(* IEC 61131-3 sources: SmartHomeNew/SmartHomeNew-main/snapshots/clean_build_2026_04_15, 26 files *)

(* ---- E_System_Root_Cause.dut ---- *)
TYPE E_System_Root_Cause :
(
    ROOT_NONE,
    ROOT_FIRE,
    ROOT_GAS_LEAK,
    ROOT_CO_WARNING,
    ROOT_CO_CRITICAL,
    ROOT_WATER_LEAK,
    ROOT_IO_OFFLINE,
    ROOT_COMM_FAULT,
    ROOT_SENSOR_FAULT,
    ROOT_SUBSYSTEM_FAULT,
    ROOT_WATCHDOG_FAULT
);
END_TYPE

(* ---- E_VENTILATION_LOCATION.dut ---- *)
{attribute 'strict'}
TYPE E_VENTILATION_LOCATION :
(
  VENT_LOCATION_NONE := 0,
  VENT_LOCATION_BASEMENT_GAME_ROOM := 1,
  VENT_LOCATION_BASEMENT_GYM := 2,
  VENT_LOCATION_BASEMENT_BOILER_ROOM := 3,
  VENT_LOCATION_BATHROOM_1F := 4,
  VENT_LOCATION_BATHROOM_2F := 5,
  VENT_LOCATION_MASTER_BATHROOM := 6,
  VENT_LOCATION_LAUNDRY := 7,
  VENT_LOCATION_KITCHEN := 8
) USINT;
END_TYPE

(* ---- ST_Heating_Command_V2.dut ---- *)
TYPE ST_Heating_Command_V2 : STRUCT
    Valve_Position_Setpoint : REAL;
END_STRUCT
END_TYPE

(* ---- ST_Lighting_Command_V2.dut ---- *)
TYPE ST_Lighting_Command_V2 : STRUCT
    Brightness_Setpoint : REAL;
END_STRUCT
END_TYPE

(* ---- ST_Maintenance_Access_Config.dut ---- *)
{attribute 'pack_mode' := '1'}
TYPE ST_Maintenance_Access_Config :
STRUCT
    maintenance_enabled : BOOL := FALSE;
    max_duration_minutes : UDINT := 60;
    requires_two_person : BOOL := TRUE;
    access_level_required : BYTE := 2;
END_STRUCT
END_TYPE

(* ---- ST_System_Diagnostics.dut ---- *)
{attribute 'pack_mode' := '1'}
TYPE ST_System_Diagnostics :
STRUCT
    Freeze_Hardware_Event_Pending : BOOL;
    Freeze_Hardware_Event_Text : STRING(200);
    Backup_Pump_Fault : BOOL;
    Electric_Heater_Fault : BOOL;
    Backup_Pump_Recovered_After_Retry : BOOL;
    Electric_Heater_Recovered_After_Retry : BOOL;
    Backup_Pump_Out_Of_Service : BOOL;
    Electric_Heater_Out_Of_Service : BOOL;

    Pump_Exercise_Active : BOOL;
    Pump_Exercise_Failed : BOOL;
    Pump_Exercise_Last_Equipment : STRING(80);
    Pump_Exercise_Last_Result : STRING(120);
    Pump_Exercise_No_Feedback_Count : INT;
    Manifold_Pump_Exercise_Count : ARRAY[1..GVL_CONSTANTS.C_MAX_MANIFOLDS] OF UDINT;
    DHW_Heating_Pump_Exercise_Count : UDINT;
    DHW_Circ_Pump_Exercise_Count : UDINT;
    Backup_Pump_Exercise_Count : UDINT;
    Pump_Exercise_Event_Seq : UDINT;
    Pump_Exercise_Journal_1 : STRING(200);
    Pump_Exercise_Journal_2 : STRING(200);
    Pump_Exercise_Journal_3 : STRING(200);
    Pump_Exercise_Journal_Last_Seq : UDINT;

    Pump_Maintenance_Required : BOOL;
    Pump_Maintenance_Warning : BOOL;

    Manifold_Pump_Out_Of_Service : ARRAY[1..GVL_CONSTANTS.C_MAX_MANIFOLDS] OF BOOL;
    DHW_Heating_Pump_Out_Of_Service : BOOL;
    DHW_Circ_Pump_Out_Of_Service : BOOL;

    Maintenance_Last_Action : STRING(120);
    Operator_Action_Blocked : BOOL;
    Operator_Block_Reason : STRING(160);
    Operator_Last_Forbidden_Action : STRING(160);
    Operator_Journal_1 : STRING(200);
    Operator_Journal_2 : STRING(200);
    Operator_Journal_3 : STRING(200);
    Operator_Journal_Event_Seq : UDINT;
    Operator_Journal_Last_Seq : UDINT;

    Dangerous_Action_Pending_Confirm : BOOL;
    Dangerous_Action_Confirm_Text : STRING(160);
    Dangerous_Action_Confirm_Deadline_MS : UDINT;
    User_Access_Level_Active : INT;
    User_Access_Denied : BOOL;
    User_Access_Deny_Reason : STRING(160);

    Valve_Test_Mode_Active : BOOL;
    Valve_Test_Deadline_MS : UDINT;
    Valve_Test_Remaining_MS : UDINT;
    Valve_Test_Validation_OK : BOOL;
    Valve_Test_Validation_Text : STRING(160);
    Valve_Test_Forced_Close : BOOL;

    Water_Valve_Test_Mode_Active : BOOL;
    Water_Valve_Test_Deadline_MS : UDINT;
    Water_Valve_Test_Remaining_MS : UDINT;
    Water_Valve_Test_Validation_OK : BOOL;
    Water_Valve_Test_Validation_Text : STRING(160);
    Water_Valve_Test_Forced_Close : BOOL;
    Gas_Valve_Test_Mode_Active : BOOL;
    Gas_Valve_Test_Deadline_MS : UDINT;
    Gas_Valve_Test_Remaining_MS : UDINT;
    Gas_Valve_Test_Validation_OK : BOOL;
    Gas_Valve_Test_Validation_Text : STRING(160);
    Gas_Valve_Test_Forced_Close : BOOL;

    Active_Leak_Sensor_Index : INT;
    Active_Gas_Sensor_Index : INT;
    Active_Leak_Zone_Name : STRING(80);
    Active_Gas_Zone_Name : STRING(80);
    Water_Valve_Test_Context : STRING(160);
    Gas_Valve_Test_Context : STRING(160);

    Water_Recovery_Target_Zone_Index : INT;
    Gas_Recovery_Target_Zone_Index : INT;
    Water_Recovery_Selective_Allowed : BOOL;
    Gas_Recovery_Selective_Allowed : BOOL;
    Water_Recovery_Selective_Text : STRING(160);
    Gas_Recovery_Selective_Text : STRING(160);
    Water_Recovery_Physical_Active : BOOL;
    Water_Recovery_Physical_Zone_Name : STRING(80);

    Water_Zone_Open_Fault : ARRAY[1..32] OF BOOL;
    Water_Zone_Close_Fault : ARRAY[1..32] OF BOOL;
    Water_Valve_Exercise_Last_Zone : INT;
    Water_Valve_Exercise_Last_Result : STRING(160);
    Water_Zone_Critical_Close_Fault : ARRAY[1..32] OF BOOL;
    Water_Close_Fault_Active : BOOL;
    Water_Close_Fault_Zone_Name : STRING(80);
    Water_Close_Fault_Text : STRING(200);
    Water_Zone_Close_Retry_Active : ARRAY[1..32] OF BOOL;
    Water_Zone_Close_Retry_Count : ARRAY[1..32] OF INT;
    Water_Zone_Close_Recovered_After_Retry : ARRAY[1..32] OF BOOL;
    Water_Localization_Failed : BOOL;
    Water_Main_Shutdown_Recommended : BOOL;
    Water_Escalation_Text : STRING(200);
    Alarm_Event_Pulse : BOOL;
    Alarm_Event_Code : UDINT;
    Alarm_Event_Value : REAL;
    Sensor_Fault : BOOL;
    IO_Offline : BOOL;
    Subsystem_Degraded : BOOL;

END_STRUCT
END_TYPE

(* ---- ST_Ventilation_Command_V2.dut ---- *)
TYPE ST_Ventilation_Command_V2 : STRUCT
    Fan_Speed_Setpoint : REAL;
END_STRUCT
END_TYPE

(* ---- GVL_CONFIG.gvl ---- *)
{attribute 'qualified_only'}
VAR_GLOBAL
    // Subsystem Configurations
    G_Heating_Config : ST_Heating_Config; // Настройки системы отопления
    G_Ventilation_Config : ST_Ventilation_Config; // Настройки системы вентиляции
    G_DHW_Config : ST_DHW_Config; // Настройки горячего водоснабжения
    G_Security_Config : ST_Security_Global_Config; // Настройки системы безопасности
    G_Flood_Config : ST_Flood_Config; // Настройки системы защиты от протечек

    // HMI Configurations
    G_HMI_FloorHeating_Configs : ARRAY[1..8] OF ST_FloorHeating_Circuit_Config; // Конфигурации контуров теплого пола
    G_Wet_Zone_Map : ARRAY[1..32] OF BOOL; // Карта мокрых зон (TRUE = мокрая зона)
    G_HMI_Tariff_Settings : ST_Tariff_Config; // Настройки тарифов
    G_HMI_Vent_Global_Config : ST_Ventilation_Global_Config; // Глобальные настройки вентиляции
    G_HMI_Vent_Unit_Configs : ARRAY[1..GVL_CONSTANTS.C_MAX_VENT_UNITS] OF ST_Ventilation_Unit_Config; // Конфигурации отдельных вентустановок
    G_HMI_Scenario_Configs : ARRAY[1..GVL_CONSTANTS.C_MAX_SCENARIOS] OF ST_Scenario_Config; // Конфигурации сценариев
    G_HMI_Outdoor_Configs : ARRAY[1..GVL_CONSTANTS.C_MAX_OUTDOOR_ZONES] OF ST_Outdoor_Zone_Config; // Конфигурации зон уличного освещения
    G_HMI_Flood_Config : ST_Flood_Global_Config; // Глобальные настройки защиты от протечек
    G_HMI_Gas_Config : ST_Gas_Valve_Configuration; // Конфигурация системы газового контроля
    G_HMI_Sensor_Calibrations : ARRAY[1..GVL_CONSTANTS.C_MAX_CALIBRATIONS] OF ST_Sensor_Calibration_Record; // Данные калибровки датчиков
    G_HMI_User_Rules : ARRAY[1..GVL_CONSTANTS.C_MAX_RULES] OF ST_User_Rule; // Пользовательские правила (Rule Engine)

    // Конфигурация тестирования клапанов
    G_Valve_Test_Config : ARRAY[1..GVL_CONSTANTS.C_MAX_MANIFOLDS] OF ST_Valve_Test_Config;

    // HMI Commands & States
    G_HMI_Cleaning_Mode_Active : ARRAY[1..GVL_CONSTANTS.C_MAX_CLEANING_MODES] OF BOOL; // Режим уборки активен
    G_HMI_Cleaning_Mode_TimeLeft : ARRAY[1..GVL_CONSTANTS.C_MAX_CLEANING_MODES] OF UINT; // Оставшееся время режима уборки
    G_HMI_Admin_2FA_Enabled : BOOL := FALSE; // Включена ли 2FA для ADMIN
    G_HMI_Current_Operator_Factor2_Done : BOOL; // Второй фактор пройден
    G_HMI_Current_Operator_ID : STRING(10); // ID текущего оператора
    G_HMI_Manual_Gas_Valve_Open : BOOL; // Ручное открытие газового клапана
    G_HMI_Manual_Gas_Valve_Time : UDINT := 5; // Время ручного открытия
    G_HMI_Manual_Gas_Valve_TimeLeft : UDINT; // Оставшееся время ручного открытия
    G_HMI_Apply_Settings : BOOL; // Команда: Применить настройки
    G_HMI_Mute_Alarm : BOOL; // Команда: Временное отключение сирены
    G_HMI_Ack_Alarms : BOOL; // Команда: Квитировать все тревоги

    // Access Control Commands
    G_HMI_Gate_Open_Req : BOOL; // Запрос на открытие въездных ворот
    G_HMI_Wicket_Open_Req : BOOL; // Запрос на открытие калитки
    G_HMI_Lock_1_Open_Req : BOOL; // Разблокировка основного замка
    G_HMI_Lock_1_Close_Req : BOOL; // Блокировка основного замка
    G_HMI_Lock_2_Open_Req : BOOL; // Разблокировка доп. замка
    G_HMI_Lock_2_Close_Req : BOOL; // Блокировка доп. замка

    // HMI Settings
    G_HMI_Language : BYTE := 0; // 0=RU, 1=EN
    G_HMI_Brightness : BYTE := 80;
    G_HMI_Screen_Saver_Timeout : UDINT := 300; // сек

    // Сетевая безопасность
    G_Allowed_IPs : ARRAY[1..GVL_CONSTANTS.C_MAX_ALLOWED_IPS] OF STRING(15) := ['192.168.1.100','192.168.1.101','127.0.0.1','','']; // Разрешенные IP-адреса для шлюза

    G_Backup_Circulation_Pump_In_Service : BOOL := TRUE; // Резервный насос доступен для логики
    G_Electric_Heater_In_Service : BOOL := TRUE; // Электронагреватель доступен для логики
    G_Freeze_Hardware_Retry_Count : INT := 2; // Количество повторных попыток для anti-freeze hardware
    G_Freeze_Hardware_Retry_Delay_MS : UDINT := 5000; // Задержка между попытками повторного пуска
    G_Pump_Exercise_Enabled : BOOL := TRUE; // Разрешение периодической прокрутки насосов после простоя
    G_Pump_Exercise_Interval_MS : UDINT := 604800000; // 7 суток
    G_Pump_Exercise_Duration_MS : UDINT := 30000; // 30 сек
    G_Manifold_Pump_In_Service : ARRAY[1..GVL_CONSTANTS.C_MAX_MANIFOLDS] OF BOOL := [TRUE, TRUE, TRUE, TRUE, TRUE];
    G_DHW_Heating_Pump_In_Service : BOOL := TRUE;
    G_DHW_Circ_Pump_In_Service : BOOL := TRUE;
    G_Water_Valve_Exercise_Enabled : BOOL := TRUE;
    G_Water_Valve_Exercise_Interval_MS : UDINT := 604800000;
    G_Water_Valve_Exercise_Duration_MS : UDINT := 15000;
    G_Water_Valve_Exercise_Window_Start : TOD := TOD#04:00;
    G_Water_Valve_Exercise_Window_End : TOD := TOD#05:00;
    G_Water_Valve_Close_Retry_Count : INT := 2;
    G_Water_Valve_Close_Retry_Delay_MS : UDINT := 3000;
    // IO Mapping
    G_FloorTemp_Map : ARRAY[1..8] OF INT := [1, 2, 3, 4, 5, 6, 7, 8];
    G_RoomTemp_Map : ARRAY[1..16] OF INT := [1, 2, 3, 4, 5, 6, 7, 8, 9, 10, 11, 12, 13, 14, 15, 16];
    G_Door_Map : ARRAY[1..GVL_CONSTANTS.C_MAX_DOOR_SENSORS] OF INT := [1, 2, 3, 4, 5, 6, 7, 8];
    G_Window_Map : ARRAY[1..16] OF INT := [9, 10, 11, 12, 13, 14, 15, 16, 17, 18, 19, 20, 21, 22, 23, 24];

    // Evacuation config
    C_MAX_LIGHT_ZONES : INT := 32; // fallback if not defined elsewhere
    G_Evac_Exit_Zones : ARRAY[1..32] OF BOOL; // зоны-выходы (TRUE = выход)
    G_Evac_Smoke_Zone_Map : ARRAY[1..GVL_CONSTANTS.C_MAX_SMOKE_SENSORS] OF INT; // Привязка дымовых датчиков к зонам эвакуации
    G_Evac_Leak_Zone_Map : ARRAY[1..GVL_CONSTANTS.C_MAX_FLOOD_SENSORS] OF INT; // Привязка датчиков протечки к зонам эвакуации
    G_Evac_Gas_Zone_Map : ARRAY[1..GVL_CONSTANTS.C_MAX_METHANE_SENSORS] OF INT; // Привязка газовых датчиков к зонам эвакуации
    G_Evac_Zone_Names : ARRAY[1..32] OF STRING(80); // Человекочитаемые имена зон (помещения/крыло/этаж/сторона)

END_VAR

VAR_GLOBAL CONSTANT
    C_MS_PER_SEC    : UDINT := GVL_CONSTANTS.C_MS_IN_SECOND; // Миллисекунд в секунде
    C_SEC_PER_MIN   : UDINT := 60; // Секунд в минуте
    C_MIN_PER_HOUR  : UDINT := 60; // Минут в часе
    C_MS_PER_MIN    : UDINT := GVL_CONSTANTS.C_MS_IN_MINUTE; // Миллисекунд в минуте
    C_MAX_RULES     : INT := 20; // Максимальное количество пользовательских правил
    C_ZONE_COUNT    : BYTE := 18; // Общее количество зон в системе

    // Коды ошибок
    ERR_PRESSURE_OUT_OF_RANGE : UDINT := 16#E004;
    ERR_HIGH_DELTA_T : UDINT := 16#E005;
    ERR_BOILER_OFFLINE : UDINT := 16#E006;
    ERR_BOILER_GENERAL_FAULT : UDINT := 16#E007;
    ERR_BOILER_NO_FLAME : UDINT := 16#E008;
    ERR_PUMP_NO_CURRENT : UDINT := 16#E009;
    ERR_PUMP_UNDERCURRENT : UDINT := 16#E00A;
    ERR_PUMP_OVERCURRENT : UDINT := 16#E00B;
    ERR_DELTA_T_LOW : UDINT := 16#E00C;
    ERR_DELTA_T_HIGH : UDINT := 16#E00D;
    ERR_DHW_IO_OFFLINE : UDINT := 16#E00E;
    ERR_DHW_TEMP_SENSOR_FAULT : UDINT := 16#E00F;
    ERR_DHW_PRESSURE_OUT_OF_RANGE : UDINT := 16#E010;
    ERR_DHW_PRESSURE_SENSOR_FAULT : UDINT := 16#E011;
END_VAR

(* ---- GVL_HEALTH_BRIDGE.gvl ---- *)
{attribute 'qualified_only'}
VAR_GLOBAL
    G_Smoke_Detected : BOOL;
    G_Gas_Detected : BOOL;
    G_Leak_Detected : BOOL;
    G_Leak_Warning_Level : BOOL;
    G_CO_Warning_Level : BOOL;
    G_CO_Alarm_Level : BOOL;
    G_Last_Fault_Event_Text : STRING(255);
END_VAR

(* ---- GVL_HEALTH_BRIDGE.st ---- *)
VAR_GLOBAL
    G_Smoke_Detected      : BOOL := FALSE;
    G_Gas_Detected        : BOOL := FALSE;
    G_CO_Warning_Level    : BOOL := FALSE;
    G_CO_Alarm_Level      : BOOL := FALSE;
    G_Leak_Detected       : BOOL := FALSE;
    G_Leak_Warning_Level  : BOOL := FALSE;

    G_Last_Fault_Event_Text : STRING(200) := '';
END_VAR

(* ---- FB_Astro_Timer.st ---- *)
FUNCTION_BLOCK FB_Astro_Timer
VAR_INPUT
    VI_System_Time_MS : UDINT;
    VI_Latitude : REAL := 55.75; // Москва (по умолчанию)
    VI_Longitude : REAL := 37.61;
    VI_Timezone : REAL := 3.0; // UTC+3
    VI_Day_Of_Year : UINT; // День года (1-365)
END_VAR
// >>> SYNC_TEST_MARKER_002 <<<
VAR_OUTPUT
    VO_Sunset_Time : TOD;
    VO_Sunrise_Time : TOD;
    VO_Is_Night : BOOL;
    VO_Current_TOD : TOD; // Текущее время суток
END_VAR
VAR
    L_Current_TOD : TOD;
    L_Pi : REAL := 3.14159265359;
    L_Rad : REAL := 3.14159265359 / 180.0;
    L_Deg : REAL := 180.0 / 3.14159265359;
    L_B : REAL;
    L_EoT : REAL;
    L_Declination : REAL;
    L_Cos_Omega : REAL;
    L_Omega : REAL;
    L_Sunrise_Local : REAL;
    L_Sunset_Local : REAL;
END_VAR

L_Current_TOD := GVL_STATUS.G_Current_TOD;
VO_Current_TOD := L_Current_TOD;

// Equation of Time (EoT) in minutes
L_B := 360.0 / 365.0 * TO_REAL(VI_Day_Of_Year - 81) * L_Rad;
L_EoT := 9.87 * SIN(2.0 * L_B) - 7.53 * COS(L_B) - 1.5 * SIN(L_B);

// Solar Declination in degrees
L_Declination := 23.45 * SIN(360.0 / 365.0 * TO_REAL(VI_Day_Of_Year + 284) * L_Rad);

// Hour angle
L_Cos_Omega := -TAN(VI_Latitude * L_Rad) * TAN(L_Declination * L_Rad);

IF L_Cos_Omega > 1.0 THEN
    L_Cos_Omega := 1.0; // Polar night
ELSIF L_Cos_Omega < -1.0 THEN
    L_Cos_Omega := -1.0; // Polar day
END_IF;

L_Omega := ACOS(L_Cos_Omega) * L_Deg;

// Sunrise and Sunset in local time (hours)
L_Sunrise_Local := 12.0 - (L_Omega / 15.0) - (L_EoT / 60.0) + (VI_Timezone * 15.0 - VI_Longitude) / 15.0;
L_Sunset_Local := 12.0 + (L_Omega / 15.0) - (L_EoT / 60.0) + (VI_Timezone * 15.0 - VI_Longitude) / 15.0;

// Handle bounds
IF L_Sunrise_Local < 0.0 THEN L_Sunrise_Local := L_Sunrise_Local + 24.0; END_IF;
IF L_Sunrise_Local >= 24.0 THEN L_Sunrise_Local := L_Sunrise_Local - 24.0; END_IF;
IF L_Sunset_Local < 0.0 THEN L_Sunset_Local := L_Sunset_Local + 24.0; END_IF;
IF L_Sunset_Local >= 24.0 THEN L_Sunset_Local := L_Sunset_Local - 24.0; END_IF;

// Конвертация в TOD
VO_Sunrise_Time := TO_TOD(TO_UDINT(L_Sunrise_Local * 3600000.0));
VO_Sunset_Time := TO_TOD(TO_UDINT(L_Sunset_Local * 3600000.0));

// ТЗ 15.2: Закат + 30 мин / Рассвет - 30 мин
VO_Is_Night := (L_Current_TOD > (VO_Sunset_Time + T#30m)) OR (L_Current_TOD < (VO_Sunrise_Time - T#30m));
// >>> SYNC_TEST_MARKER_FORCE <<<
// >>> BULK_SYNC_ANCHOR: FB_Astro_Timer <<<

(* ---- FB_DHW_Manager.st ---- *)
FUNCTION_BLOCK FB_DHW_Manager
VAR_INPUT
    VI_System_Time_MS : UDINT; // Системное время (мс)
    VI_Current_TOD : TOD; // Текущее время суток
    VI_IsActivePLC : BOOL; // Флаг: Данный ПЛК является ведущим
    VI_Temp : REAL; // Текущая температура воды в бойлере (°C)
    VI_Pressure : REAL; // Текущее давление в системе ГВС (бар)
    VI_Config : ST_DHW_Config; // Конфигурация системы ГВС (уставки, расписание)
    VI_Current_Day_Of_Week : UINT; // Текущий день недели (1-7)
    VI_Reset_Errors : BOOL; // Сброс ошибок
    VI_Emergency_Stop : BOOL; // Агрегированный аварийный стоп от подсистемы безопасности
    VI_System_Mode : E_System_Operating_Mode; // Агрегированный режим системы
    VI_IO_Modules_Online : ARRAY[1..GVL_CONSTANTS.C_MAX_MODULES] OF BOOL; // Статусы модулей ввода-вывода (только чтение)
END_VAR
// >>> SYNC_TEST_MARKER_001 <<<
VAR_OUTPUT
    VO_Status : ST_DHW_Status; // Сводный статус системы ГВС для HMI
    VO_Heating_Pump : BOOL; // Выход: Управление насосом нагрева (загрузка бойлера)
    VO_Circ_Pump : BOOL; // Выход: Управление насосом рециркуляции ГВС
END_VAR
VAR
    // DHW V2 staging layer
    fbDHWV2Staging : FB_DHW_V2_Staging;
    L_DHW_V2_Command_V2 : ST_DHW_Command_V2;
    L_DHW_V2_State_V2 : ST_DHW_State_V2;
    L_DHW_V2_Shadow_Diff_Found : BOOL;
    L_DHW_V2_Switch_Enabled : BOOL;
    L_DHW_V2_Path_Ready : BOOL;
    L_DHW_Using_Legacy_Fallback : BOOL;
    L_i : INT;
    L_Current_TOD : TOD; // Текущее время суток
    L_Legionella_Active : BOOL; // Флаг активного режима термической дезинфекции (Легионелла)
    L_Legionella_Timer : FB_System_Timer; // Таймер удержания температуры для дезинфекции
    L_Last_Good_Temp : REAL := 55.0; // Последнее достоверное значение температуры (для Fallback)
    L_Legionella_Done_Today : BOOL; // Признак выполнения термодезинфекции в текущие сутки
    L_Last_Legionella_Day : UINT; // День недели последнего сброса/контроля цикла легионеллы
    fbTempValidator : FB_Analog_Validator;
    fbPressValidator : FB_Analog_Validator;
    L_Error_Latched : BOOL;
    L_Error_ID_Latched : WORD;
    L_Policy_Degraded : BOOL;
    L_Policy_Freeze_Protection : BOOL;
    L_Policy_Safe_Stop : BOOL;
    L_Target_Temp_Adjusted : REAL;
END_VAR

IF NOT VI_IsActivePLC THEN RETURN; END_IF;

L_DHW_V2_Shadow_Diff_Found := FALSE;
L_DHW_V2_Switch_Enabled := TRUE;
L_DHW_V2_Path_Ready := FALSE;
L_DHW_Using_Legacy_Fallback := TRUE;

GVL_STATE.G_DHW_IO_Fault := FALSE;
GVL_STATE.G_DHW_Sensor_Fault := FALSE;
GVL_STATE.G_DHW_Subsystem_Degraded := FALSE;

IF VI_Emergency_Stop THEN
    VO_Heating_Pump := FALSE;
    VO_Circ_Pump := FALSE;
    VO_Status.Warning := FALSE;
    VO_Status.Error := TRUE;
    VO_Status.Error_ID := TO_WORD(GVL_CONFIG.ERR_DHW_IO_OFFLINE); // временно используем общий аварийный код до детализации safety-кодов
    VO_Status.Heating_Pump_On := FALSE;
    VO_Status.Circ_Pump_On := FALSE;
    RETURN;
END_IF;

// Фиксация текущего времени
L_Current_TOD := VI_Current_TOD;

// ========================================
// DHW POLICY LAYER
// ========================================
L_Policy_Safe_Stop := (VI_System_Mode = E_System_Operating_Mode.MODE_SAFE_STOP);
L_Policy_Freeze_Protection := (VI_System_Mode = E_System_Operating_Mode.MODE_FREEZE_PROTECTION);
L_Policy_Degraded := (VI_System_Mode = E_System_Operating_Mode.MODE_DEGRADED);
L_Target_Temp_Adjusted := VI_Config.Target_Temp;
IF L_Policy_Degraded THEN
    L_Target_Temp_Adjusted := VI_Config.Target_Temp - VI_Config.Degraded_Target_Delta;
END_IF;

// ========================================
// DHW POLICY OVERRIDE
// ========================================
IF L_Policy_Safe_Stop THEN
    VO_Heating_Pump := FALSE;
    VO_Circ_Pump := FALSE;
    RETURN;
END_IF;

IF L_Policy_Freeze_Protection THEN
    VO_Heating_Pump := FALSE;
    VO_Circ_Pump := FALSE;
    RETURN;
END_IF;

// Сброс признака выполнения термодезинфекции при смене дня.
IF L_Last_Legionella_Day <> VI_Current_Day_Of_Week THEN
    L_Legionella_Done_Today := FALSE;
    L_Last_Legionella_Day := VI_Current_Day_Of_Week;
END_IF;

// Базовый сброс незащёлкнутых статусных флагов на текущий цикл.
// Критические ошибки ниже могут зафиксироваться и завершить выполнение через RETURN.
VO_Status.Warning := FALSE;
VO_Status.Error := FALSE;
VO_Status.Error_ID := 0;

// Сброс ошибок
IF VI_Reset_Errors THEN
    L_Error_Latched := FALSE;
    L_Error_ID_Latched := 0;
END_IF;

// Проверка связи с модулями ввода-вывода
FOR L_i := 1 TO GVL_CONSTANTS.C_MAX_MODULES DO
    IF NOT VI_IO_Modules_Online[L_i] THEN
        L_Error_Latched := TRUE;
        GVL_STATE.G_DHW_IO_Fault := TRUE;
        L_Error_ID_Latched := TO_WORD(GVL_CONFIG.ERR_DHW_IO_OFFLINE); // Потеря связи с модулями ввода-вывода
    END_IF;
END_FOR;

// 1. Обработка неисправностей датчиков и сервисных режимов (ТЗ 7.0)
fbTempValidator(
    VI_Value := VI_Temp,
    VI_Min_Valid := 0.0,
    VI_Max_Valid := 100.0,
    VI_Fallback_Mode := 0,
    VI_Default_Value := 55.0
);

fbPressValidator(
    VI_Value := VI_Pressure,
    VI_Min_Valid := 0.0,
    VI_Max_Valid := 10.0,
    VI_Fallback_Mode := 0
);

VO_Status.Temp := fbTempValidator.VO_Value;
VO_Status.Pressure := fbPressValidator.VO_Value;

// Сохраняем последнее достоверное значение температуры ГВС.
// Используется только для диагностики/сервиса, не для fallback-управления.
IF NOT fbTempValidator.VO_Error THEN
    L_Last_Good_Temp := VO_Status.Temp;
END_IF;

IF fbTempValidator.VO_Error THEN
    GVL_STATE.G_DHW_Sensor_Fault := TRUE;
    L_Error_Latched := TRUE;
    L_Error_ID_Latched := TO_WORD(GVL_CONFIG.ERR_DHW_TEMP_SENSOR_FAULT); // Критическая ошибка датчика температуры
ELSIF (VO_Status.Pressure < 1.0 OR VO_Status.Pressure > 4.0) AND NOT fbPressValidator.VO_Error THEN
    L_Error_Latched := TRUE;
    L_Error_ID_Latched := TO_WORD(GVL_CONFIG.ERR_DHW_PRESSURE_OUT_OF_RANGE); // Давление вне нормы
END_IF;

IF L_Error_Latched THEN
    // Критическая ошибка: переход в безопасное состояние с полной остановкой насосов.
    VO_Heating_Pump := FALSE;
    VO_Circ_Pump := FALSE;
    VO_Status.Warning := FALSE;
    VO_Status.Error := TRUE;
    VO_Status.Error_ID := L_Error_ID_Latched;
    VO_Status.Heating_Pump_On := FALSE;
    VO_Status.Circ_Pump_On := FALSE;
    RETURN;
END_IF;

// Ошибка датчика давления не останавливает ГВС,
// но переводит подсистему в режим предупреждения (degraded mode).
IF fbPressValidator.VO_Error THEN
    GVL_STATE.G_DHW_Sensor_Fault := TRUE;
    GVL_STATE.G_DHW_Subsystem_Degraded := TRUE;
    VO_Status.Warning := TRUE;
    VO_Status.Error := FALSE;
    VO_Status.Error_ID := TO_WORD(GVL_CONFIG.ERR_DHW_PRESSURE_SENSOR_FAULT);
END_IF;

// 2. Логика поддержания температуры воды в бойлере (Нагрев)
// На этом этапе FB уже выполняется только на активном ПЛК.

// Термическая дезинфекция (Легионелла)
IF VI_Config.Anti_Legionella_Enabled
   AND (VI_Current_Day_Of_Week = VI_Config.Anti_Legionella_Day)
   AND (L_Current_TOD >= TOD#02:00)
   AND (L_Current_TOD <= TOD#04:00)
   AND NOT L_Legionella_Done_Today THEN
    L_Legionella_Active := TRUE;
ELSE
    L_Legionella_Active := FALSE;
END_IF;

L_Legionella_Timer(IN := L_Legionella_Active AND VO_Status.Temp >= 70.0, PT := T#30m, VI_System_Time_MS := VI_System_Time_MS);
IF L_Legionella_Timer.Q THEN
    L_Legionella_Active := FALSE; // Дезинфекция завершена
    L_Legionella_Done_Today := TRUE; // Повторно в те же сутки не запускать
END_IF;

// Двухпозиционное регулирование с гистерезисом
IF L_Legionella_Active THEN
    IF VO_Status.Temp < 70.0 THEN
        VO_Heating_Pump := TRUE;
    ELSIF VO_Status.Temp > 72.0 THEN
        VO_Heating_Pump := FALSE;
    END_IF;
ELSE
    IF VO_Status.Temp < (L_Target_Temp_Adjusted - VI_Config.Hysteresis) THEN
        VO_Heating_Pump := TRUE;
    ELSIF VO_Status.Temp > (L_Target_Temp_Adjusted + VI_Config.Hysteresis) THEN
        VO_Heating_Pump := FALSE;
    END_IF;
END_IF;

// 3. Управление циркуляционным насосом ГВС по расписанию
// Рециркуляция обеспечивает мгновенное наличие горячей воды у потребителя
VO_Circ_Pump := SEL(VI_Config.Circulation_Schedule_Enabled AND NOT (VI_Config.Night_Mode_Enabled AND (L_Current_TOD < VI_Config.Circulation_Start OR L_Current_TOD > VI_Config.Circulation_End)), FALSE, TRUE);

// Формирование статусных данных для визуализации.
// К этому моменту статус уже консистентен:
// - Error = критическая ошибка с остановкой ГВС
// - Warning = деградация без остановки
VO_Status.Heating_Pump_On := VO_Heating_Pump;
VO_Status.Circ_Pump_On := VO_Circ_Pump;

// ========================================
// DHW V2 staging execution
// ========================================
fbDHWV2Staging(
    VI_Tank_ID := 1,
    VI_Enable := TRUE,
    VI_Target_Temp := VI_Config.Target_Temp,
    VI_Pump_Enable := VO_Heating_Pump,
    VI_Heating_Priority := FALSE,

    VI_Is_Active := TRUE,
    VI_Tank_Temp := VO_Status.Temp,
    VI_Supply_Temp := VO_Status.Temp,
    VI_Return_Temp := VO_Status.Temp,
    VI_Pump_Actual := VO_Heating_Pump,
    VI_Alarm_Active := VO_Status.Error,

    VO_Command_Shadow => L_DHW_V2_Command_V2,
    VO_State_Shadow => L_DHW_V2_State_V2
);

// ========================================
// DHW V2 staging validation
// ========================================
IF VO_Heating_Pump <> (L_DHW_V2_Command_V2.Pump_Enable > 0.5) THEN
    L_DHW_V2_Shadow_Diff_Found := TRUE;
END_IF;
IF ABS(VO_Status.Temp - L_DHW_V2_State_V2.Tank_Temp) > 0.1 THEN
    L_DHW_V2_Shadow_Diff_Found := TRUE;
END_IF;
IF ABS(VO_Status.Pressure - L_DHW_V2_State_V2.Supply_Temp) > 0.1 THEN
    L_DHW_V2_Shadow_Diff_Found := TRUE;
END_IF;

// Guarded DHW V2 enable
IF L_DHW_V2_Switch_Enabled THEN
    IF NOT L_DHW_V2_Shadow_Diff_Found THEN
        L_DHW_V2_Path_Ready := TRUE;
        L_DHW_Using_Legacy_Fallback := FALSE;
    ELSE
        L_DHW_V2_Path_Ready := FALSE;
        L_DHW_Using_Legacy_Fallback := TRUE;
    END_IF;
ELSE
    L_DHW_V2_Path_Ready := FALSE;
    L_DHW_Using_Legacy_Fallback := TRUE;
END_IF;

END_FUNCTION_BLOCK
// >>> BULK_SYNC_ANCHOR: FB_DHW_Manager <<<

(* ---- FB_Exhaust_Ventilation_Controller.st ---- *)
FUNCTION_BLOCK FB_Exhaust_Ventilation_Controller
VAR_INPUT
    VI_Humidity : REAL;
    VI_CO2      : REAL;
    VI_Config   : ST_Ventilation_Unit_Config;
END_VAR
VAR_OUTPUT
    VO_Fan_Speed : BYTE;
END_VAR

IF VI_Humidity > VI_Config.Threshold_Hum THEN
    VO_Fan_Speed := 100;
ELSIF VI_CO2 > 800.0 THEN
    VO_Fan_Speed := 70;
ELSE
    VO_Fan_Speed := 40;
END_IF;

(* ---- FB_Gas_Methane_Detector.st ---- *)
FUNCTION_BLOCK FB_Gas_Methane_Detector
VAR_INPUT
    VI_Methane_LEL : REAL;
    VI_Threshold   : REAL := 20.0;
END_VAR
VAR_OUTPUT
    VO_Gas_Detected : BOOL;
END_VAR

VO_Gas_Detected := (VI_Methane_LEL >= VI_Threshold);

(* ---- FB_Gas_Smoke_Manager.st ---- *)
FUNCTION_BLOCK FB_Gas_Smoke_Manager
VAR_INPUT
    VI_System_Time_MS : UDINT;
    VI_IsActivePLC    : BOOL;
    VI_Mute_Request   : BOOL;
END_VAR

VAR_IN_OUT
    VI_Methane_LEL    : ARRAY[1..GVL_CONSTANTS.C_MAX_METHANE_SENSORS] OF REAL;
    VI_CO_PPM         : ARRAY[1..GVL_CONSTANTS.C_MAX_CO_SENSORS] OF REAL;
    VI_Smoke_Sensors  : ARRAY[1..GVL_CONSTANTS.C_MAX_SMOKE_SENSORS] OF BOOL;
END_VAR

VAR_OUTPUT
    // Health signals
    VO_Smoke_Detected   : BOOL;
    VO_Gas_Detected     : BOOL;
    VO_CO_Warning_Level : BOOL;
    VO_CO_Alarm_Level   : BOOL;

    // Actuators
    VO_Siren_Active      : BOOL;
    VO_Gas_Valve_Close   : BOOL;
    VO_Boiler_Stop       : BOOL;
    VO_Vent_PV3_Boost    : BOOL;
    VO_Supply_100_Req    : BOOL;
    VO_Exhaust_100_Req   : BOOL;
    VO_Supply_80_Req     : BOOL;
    VO_Vent_Stop         : BOOL;

    VO_Status_Msg        : STRING(200);
END_VAR

VAR
    L_Methane_Max   : REAL;
    L_CO_Max        : REAL;
    L_Smoke_Count   : UINT;
    L_Smoke_Active  : BOOL;
    L_i             : INT;

    L_CO_Timer_30ppm  : FB_System_Timer;
    L_CO_Timer_70ppm  : FB_System_Timer;
    L_CO_Timer_400ppm : FB_System_Timer;

    L_CO_Level_30   : BOOL;
    L_CO_Level_70   : BOOL;
    L_CO_Level_400  : BOOL;

    L_Smoke_Timer : ARRAY[1..GVL_CONSTANTS.C_MAX_SMOKE_SENSORS] OF FB_System_Timer;
END_VAR

IF NOT VI_IsActivePLC THEN RETURN; END_IF;

// Reset outputs
VO_Smoke_Detected := FALSE;
VO_Gas_Detected := FALSE;
VO_CO_Warning_Level := FALSE;
VO_CO_Alarm_Level := FALSE;

VO_Siren_Active := FALSE;
VO_Gas_Valve_Close := FALSE;
VO_Boiler_Stop := FALSE;
VO_Vent_PV3_Boost := FALSE;
VO_Supply_100_Req := FALSE;
VO_Exhaust_100_Req := FALSE;
VO_Supply_80_Req := FALSE;
VO_Vent_Stop := FALSE;
VO_Status_Msg := 'ОК';

// --- Methane ---
L_Methane_Max := 0.0;
FOR L_i := 1 TO GVL_CONSTANTS.C_MAX_METHANE_SENSORS DO
    IF VI_Methane_LEL[L_i] > L_Methane_Max THEN
        L_Methane_Max := VI_Methane_LEL[L_i];
    END_IF;
END_FOR;

IF L_Methane_Max >= 10.0 THEN
    VO_Vent_PV3_Boost := TRUE;
END_IF;

IF L_Methane_Max >= 20.0 THEN
    VO_Gas_Detected := TRUE;
    VO_Gas_Valve_Close := TRUE;
    VO_Boiler_Stop := TRUE;
    VO_Supply_100_Req := TRUE;
END_IF;

// --- CO ---
L_CO_Max := 0.0;
FOR L_i := 1 TO GVL_CONSTANTS.C_MAX_CO_SENSORS DO
    IF VI_CO_PPM[L_i] > L_CO_Max THEN
        L_CO_Max := VI_CO_PPM[L_i];
    END_IF;
END_FOR;

L_CO_Level_30 := (L_CO_Max >= 30.0);
L_CO_Level_70 := (L_CO_Max >= 70.0);
L_CO_Level_400 := (L_CO_Max >= 400.0);

L_CO_Timer_30ppm(IN := L_CO_Level_30, PT := T#8h, VI_System_Time_MS := VI_System_Time_MS);
L_CO_Timer_70ppm(IN := L_CO_Level_70, PT := T#1h, VI_System_Time_MS := VI_System_Time_MS);
L_CO_Timer_400ppm(IN := L_CO_Level_400, PT := T#15m, VI_System_Time_MS := VI_System_Time_MS);

IF L_CO_Timer_30ppm.Q THEN
    VO_CO_Warning_Level := TRUE;
    VO_Supply_80_Req := TRUE;
END_IF;

IF L_CO_Timer_70ppm.Q OR L_CO_Timer_400ppm.Q THEN
    VO_CO_Alarm_Level := TRUE;
    VO_Supply_80_Req := TRUE;
END_IF;

// --- Smoke ---
L_Smoke_Count := 0;
L_Smoke_Active := FALSE;

FOR L_i := 1 TO GVL_CONSTANTS.C_MAX_SMOKE_SENSORS DO
    L_Smoke_Timer[L_i](IN := VI_Smoke_Sensors[L_i], PT := T#30s, VI_System_Time_MS := VI_System_Time_MS);

    IF VI_Smoke_Sensors[L_i] THEN
        L_Smoke_Count := L_Smoke_Count + 1;
    END_IF;

    IF L_Smoke_Timer[L_i].Q OR (L_Smoke_Count >= 2) THEN
        L_Smoke_Active := TRUE;
    END_IF;
END_FOR;

IF L_Smoke_Active THEN
    VO_Smoke_Detected := TRUE;
    VO_Vent_Stop := TRUE;
    VO_Boiler_Stop := TRUE;
END_IF;

// Status
IF VO_Smoke_Detected THEN
    VO_Status_Msg := 'ПОЖАР';
ELSIF VO_Gas_Detected THEN
    VO_Status_Msg := 'УТЕЧКА ГАЗА';
ELSIF VO_CO_Alarm_Level THEN
    VO_Status_Msg := 'КРИТИЧЕСКИЙ CO';
ELSIF VO_CO_Warning_Level THEN
    VO_Status_Msg := 'ПОВЫШЕННЫЙ CO';
ELSE
    VO_Status_Msg := 'ОК';
END_IF;
// >>> BULK_SYNC_ANCHOR: FB_Gas_Smoke_Manager <<<

(* ---- FB_Gateway_Interface.st ---- *)
FUNCTION_BLOCK FB_Gateway_Interface
VAR_INPUT
    VI_System_Time_MS           : UDINT;
    VI_Local_PLC_Role           : E_PLC_ROLE;
    VI_Incoming_Command         : ST_Gateway_Command;
    VI_Command_Received         : BOOL;

    // Состояния системы
    VI_Outdoor_Temp             : REAL;
    VI_Security_Armed           : BOOL;
    VI_Flood_Alarm_Active       : BOOL;
    VI_Gas_Alarm_Active         : BOOL;
    VI_Fire_Alarm_Active        : BOOL;
    VI_Methane_Concentration    : REAL;
    VI_Active_Scenario          : E_SCENARIO_TYPE;

    // 2FA
    VI_Send_2FA_Req             : BOOL;
    VI_2FA_Code                 : STRING(6);

    // Конфигурация
END_VAR
VAR_IN_OUT
    VI_FloorHeating_Temps       : ARRAY[1..8] OF REAL;
    VI_Room_Temps               : ARRAY[1..16] OF REAL;
    VI_Zone_Valve_States        : ARRAY[1..8] OF BOOL;
    VI_Manifold_Pressures       : ARRAY[1..GVL_CONSTANTS.C_MAX_MANIFOLDS] OF REAL;
    VI_Manifold_Pump_States     : ARRAY[1..GVL_CONSTANTS.C_MAX_MANIFOLDS] OF BOOL;
    VI_Lighting_Base_Levels     : ARRAY[1..32] OF BYTE;
    VI_Socket_States            : ARRAY[1..GVL_CONSTANTS.C_MAX_SOCKETS] OF BOOL;
    VI_Blinds_Positions         : ARRAY[1..GVL_CONSTANTS.C_MAX_BLINDS] OF BYTE;
    VI_Allowed_IPs              : ARRAY[1..GVL_CONSTANTS.C_MAX_ALLOWED_IPS] OF STRING(15);
END_VAR

VAR_OUTPUT
    VO_Modbus_Registers         : ARRAY[0..GVL_CONSTANTS.C_MAX_MODBUS_REGISTERS-1] OF WORD; // Расширенный диапазон
    VO_Lighting_Override        : ARRAY[1..32] OF BYTE;
    VO_Blinds_Override          : ARRAY[1..GVL_CONSTANTS.C_MAX_BLINDS] OF BYTE;
    VO_Socket_Override          : ARRAY[1..GVL_CONSTANTS.C_MAX_SOCKETS] OF BOOL;
    VO_Arm_Req                  : BOOL;
    VO_Disarm_Req               : BOOL;
    VO_PIN_Code                 : STRING(4);
    VO_RFID_Tag                 : STRING(20);
    VO_2FA_Code_In              : STRING(6);
    VO_Data_Ready               : BOOL;
    VO_HMI_Status_Message       : STRING(200);
    VO_Telegram_Msg             : STRING(200);
    VO_Send_Telegram            : BOOL;

    // Выходы для управления конфигурацией и состоянием
    VO_Set_Scenario_Req         : BOOL;
    VO_Target_Scenario          : E_SCENARIO_TYPE;
    VO_Set_Temp_Req             : BOOL;
    VO_Target_Zone              : INT;
    VO_Target_Temp              : REAL;
    VO_Set_Vent_Req             : BOOL;
    VO_Target_Vent_Speed        : BYTE;
    VO_Reset_Errors_Req         : BOOL; // Запрос на сброс ошибок/квитирование
    VO_Set_Config_Req           : BOOL; // Запрос на применение конфигурации
    VO_Sync_Time_Req            : BOOL; // Запрос на синхронизацию времени
    VO_New_Time_MS              : UDINT; // Новое время (мс с начала суток)
END_VAR

VAR
    L_last_update_time          : UDINT;
    L_i                         : INT;
    L_j                         : INT;
    L_idx                       : INT;
    L_tmp_word                  : WORD;
    L_Code_UDINT                : UDINT;
    L_Prev_Fire                 : BOOL;
    L_Prev_Gas                  : BOOL;
    L_Prev_Flood                : BOOL;
    L_Prev_Security             : BOOL;
    L_Deduplicator              : FB_Command_Deduplication;
    L_CRC_Calc                  : FB_CRC32_Calculator;
    L_Calculated_CRC            : DWORD;
    L_Command_Size              : UDINT;
    L_IP_Allowed                : BOOL;

    L_Process_Command           : ST_Gateway_Command;
    L_Has_Command_To_Process    : BOOL;
END_VAR

VAR RETAIN
    // Буфер команд для резервного ПЛК
    L_Command_Buffer            : ARRAY[1..GVL_CONSTANTS.C_MAX_GATEWAY_COMMANDS] OF ST_Gateway_Command;
    L_Buffer_Head               : INT := 1;
    L_Buffer_Tail               : INT := 1;
    L_Buffer_Count              : INT := 0;
END_VAR

// Отправка уведомлений в Telegram (ТЗ 10.2)
VO_Send_Telegram := FALSE;
IF VI_Fire_Alarm_Active AND NOT L_Prev_Fire THEN
    VO_Telegram_Msg := 'ВНИМАНИЕ! ПОЖАРНАЯ ТРЕВОГА!';
    VO_Send_Telegram := TRUE;
END_IF;
IF VI_Gas_Alarm_Active AND NOT L_Prev_Gas THEN
    VO_Telegram_Msg := 'ВНИМАНИЕ! УТЕЧКА ГАЗА!';
    VO_Send_Telegram := TRUE;
END_IF;
IF VI_Flood_Alarm_Active AND NOT L_Prev_Flood THEN
    VO_Telegram_Msg := 'ВНИМАНИЕ! ПРОТЕЧКА ВОДЫ!';
    VO_Send_Telegram := TRUE;
END_IF;
IF VI_Security_Armed AND NOT L_Prev_Security THEN
    VO_Telegram_Msg := 'ОХРАНА ВКЛЮЧЕНА';
    VO_Send_Telegram := TRUE;
ELSIF NOT VI_Security_Armed AND L_Prev_Security THEN
    VO_Telegram_Msg := 'ОХРАНА ОТКЛЮЧЕНА';
    VO_Send_Telegram := TRUE;
END_IF;

L_Prev_Fire := VI_Fire_Alarm_Active;
L_Prev_Gas := VI_Gas_Alarm_Active;
L_Prev_Flood := VI_Flood_Alarm_Active;
L_Prev_Security := VI_Security_Armed;

// Обновление данных Modbus (раз в 1 сек)
IF (VI_System_Time_MS - L_last_update_time) >= GVL_CONSTANTS.C_MS_IN_SECOND THEN
    L_last_update_time := VI_System_Time_MS;

    // 0: Статус ПЛК и Аварии
    L_tmp_word := 0;
    IF VI_Local_PLC_Role = E_PLC_ROLE.ROLE_ACTIVE THEN L_tmp_word := L_tmp_word OR 1; END_IF;
    IF VI_Security_Armed THEN L_tmp_word := L_tmp_word OR 2; END_IF;
    IF VI_Flood_Alarm_Active THEN L_tmp_word := L_tmp_word OR 4; END_IF;
    IF VI_Gas_Alarm_Active THEN L_tmp_word := L_tmp_word OR 8; END_IF;
    IF VI_Fire_Alarm_Active THEN L_tmp_word := L_tmp_word OR 16; END_IF;
    VO_Modbus_Registers[0] := L_tmp_word;

    // 1-16: Температуры пола (x10)
    FOR L_i := 1 TO 8 DO
        VO_Modbus_Registers[L_i] := TO_WORD(TO_INT(VI_FloorHeating_Temps[L_i] * 10.0));
    END_FOR;

    // 17-310102: Температуры помещений (x10)
    FOR L_i := 1 TO 16 DO
        VO_Modbus_Registers[16 + L_i] := TO_WORD(TO_INT(VI_Room_Temps[L_i] * 10.0));
    END_FOR;

    // 310103: Состояние клапанов зон (битовая маска 1-16)
    L_tmp_word := 0;
    FOR L_i := 1 TO 8 DO
        IF VI_Zone_Valve_States[L_i] THEN
            L_tmp_word := L_tmp_word OR SHL(TO_WORD(1), L_i - 1);
        END_IF;
    END_FOR;
    VO_Modbus_Registers[33] := L_tmp_word;

    // 34-38: Давление в коллекторах (x100)
    FOR L_i := 1 TO GVL_CONSTANTS.C_MAX_MANIFOLDS DO
        VO_Modbus_Registers[33 + L_i] := TO_WORD(TO_INT(VI_Manifold_Pressures[L_i] * 100.0));
    END_FOR;

    // 40-55: Базовое освещение
    FOR L_i := 1 TO 32 DO
        VO_Modbus_Registers[39 + L_i] := TO_WORD(VI_Lighting_Base_Levels[L_i]);
    END_FOR;

    // 60-79: Положение штор (20 шт)
    FOR L_i := 1 TO GVL_CONSTANTS.C_MAX_BLINDS DO
        VO_Modbus_Registers[59 + L_i] := TO_WORD(VI_Blinds_Positions[L_i]);
    END_FOR;

    // 80-82: Розетки (битовая маска, 36 розеток -> 3 WORD)
    FOR L_i := 0 TO (GVL_CONSTANTS.C_MAX_SOCKETS - 1) / 16 DO
        L_tmp_word := 0;
        FOR L_j := 1 TO 16 DO
            L_idx := (L_i * 16) + L_j;
            IF L_idx <= GVL_CONSTANTS.C_MAX_SOCKETS THEN
                IF VI_Socket_States[L_idx] THEN
                    L_tmp_word := L_tmp_word OR SHL(TO_WORD(1), L_j - 1);
                END_IF;
            END_IF;
        END_FOR;
        VO_Modbus_Registers[79 + L_i] := L_tmp_word;
    END_FOR;

    // 100-102: 2FA Request and Code
    VO_Modbus_Registers[100] := SEL(VI_Send_2FA_Req, 0, 1);
    IF VI_Send_2FA_Req THEN
        L_Code_UDINT := STRING_TO_UDINT(VI_2FA_Code);
        VO_Modbus_Registers[101] := TO_WORD(L_Code_UDINT AND 16#FFFF);
        VO_Modbus_Registers[102] := TO_WORD(SHR(L_Code_UDINT, 16));
    ELSE
        VO_Modbus_Registers[101] := 0;
        VO_Modbus_Registers[102] := 0;
    END_IF;

    VO_Data_Ready := TRUE;
END_IF;

// Обработка входящих команд
VO_Arm_Req := FALSE;
VO_Disarm_Req := FALSE;
VO_Set_Scenario_Req := FALSE;
VO_Set_Temp_Req := FALSE;
VO_Set_Vent_Req := FALSE;
VO_Reset_Errors_Req := FALSE;
VO_Set_Config_Req := FALSE;
VO_Sync_Time_Req := FALSE;
L_Has_Command_To_Process := FALSE;

// 1. Прием команды и буферизация
IF VI_Command_Received THEN
    IF VI_Local_PLC_Role = E_PLC_ROLE.ROLE_ACTIVE THEN
        // Если активен, обрабатываем сразу
        L_Process_Command := VI_Incoming_Command;
        L_Has_Command_To_Process := TRUE;
    ELSE
        // Если резервный, добавляем в буфер
        IF L_Buffer_Count < GVL_CONSTANTS.C_MAX_GATEWAY_COMMANDS THEN
            L_Command_Buffer[L_Buffer_Head] := VI_Incoming_Command;
            L_Buffer_Head := L_Buffer_Head + 1;
            IF L_Buffer_Head > GVL_CONSTANTS.C_MAX_GATEWAY_COMMANDS THEN L_Buffer_Head := 1; END_IF;
            L_Buffer_Count := L_Buffer_Count + 1;
        END_IF;
    END_IF;
END_IF;

// 2. Извлечение из буфера при переходе в активный режим
IF NOT L_Has_Command_To_Process AND (VI_Local_PLC_Role = E_PLC_ROLE.ROLE_ACTIVE) AND (L_Buffer_Count > 0) THEN
    L_Process_Command := L_Command_Buffer[L_Buffer_Tail];
    L_Buffer_Tail := L_Buffer_Tail + 1;
    IF L_Buffer_Tail > GVL_CONSTANTS.C_MAX_GATEWAY_COMMANDS THEN L_Buffer_Tail := 1; END_IF;
    L_Buffer_Count := L_Buffer_Count - 1;
    L_Has_Command_To_Process := TRUE;
END_IF;

// 3. Обработка команды
IF L_Has_Command_To_Process THEN
    // Проверка IP-адреса источника
    L_IP_Allowed := FALSE;
    IF L_Process_Command.source_ip = '' THEN
        L_IP_Allowed := TRUE; // Если IP не передан, пропускаем (для обратной совместимости или локальных вызовов)
    ELSE
        FOR L_i := 1 TO GVL_CONSTANTS.C_MAX_ALLOWED_IPS DO
            IF VI_Allowed_IPs[L_i] = L_Process_Command.source_ip THEN
                L_IP_Allowed := TRUE;
                EXIT;
            END_IF;
        END_FOR;
    END_IF;

    IF NOT L_IP_Allowed THEN
        VO_HMI_Status_Message := 'Gateway: Ошибка безопасности (Неизвестный IP)';
        RETURN;
    END_IF;

    // Проверка целостности данных (CRC32)
    // Размер данных для расчета CRC: размер структуры минус размер самого поля crc32
    L_Command_Size := SIZEOF(L_Process_Command) - SIZEOF(L_Process_Command.crc32);
    L_Calculated_CRC := L_CRC_Calc.Calculate();

    IF L_Calculated_CRC = L_Process_Command.crc32 THEN
        L_Deduplicator(
            VI_Command_ID := L_Process_Command.command_id,
            VI_Command_Type := L_Process_Command.command_type,
            VI_Command_Value := L_Process_Command.target_value,
            VI_System_Time_MS := VI_System_Time_MS
        );

        IF L_Deduplicator.VO_Is_New_Command THEN
            CASE L_Process_Command.command_type OF
        E_Gateway_Command_Type.CMD_SET_SCENARIO: // Управление сценариями
            VO_Set_Scenario_Req := TRUE;
            VO_Target_Scenario := L_Process_Command.target_scenario;
            VO_HMI_Status_Message := 'Gateway: Сценарий изменен';
        E_Gateway_Command_Type.CMD_SET_LIGHT: // Управление освещением
            IF (L_Process_Command.target_zone >= 1) AND (L_Process_Command.target_zone <= 32) THEN
                VO_Lighting_Override[L_Process_Command.target_zone] := TO_BYTE(L_Process_Command.target_value);
                VO_HMI_Status_Message := 'Gateway: Команда освещения принята';
            END_IF;
        E_Gateway_Command_Type.CMD_SET_BLINDS: // Управление шторами
            IF (L_Process_Command.target_zone >= 1) AND (L_Process_Command.target_zone <= GVL_CONSTANTS.C_MAX_BLINDS) THEN
                VO_Blinds_Override[L_Process_Command.target_zone] := TO_BYTE(L_Process_Command.target_value);
                VO_HMI_Status_Message := 'Gateway: Команда штор принята';
            END_IF;
        E_Gateway_Command_Type.CMD_SET_SOCKET: // Розетки
            IF (L_Process_Command.target_zone >= 1) AND (L_Process_Command.target_zone <= GVL_CONSTANTS.C_MAX_SOCKETS) THEN
                VO_Socket_Override[L_Process_Command.target_zone] := L_Process_Command.target_on_off;
                VO_HMI_Status_Message := 'Gateway: Команда розетки принята';
            END_IF;
        E_Gateway_Command_Type.CMD_SET_SECURITY: // Охрана
            IF L_Process_Command.target_armed THEN
                VO_Arm_Req := TRUE;
            ELSE
                VO_Disarm_Req := TRUE;
            END_IF;
            VO_PIN_Code := L_Process_Command.target_pin;
            VO_2FA_Code_In := L_Process_Command.target_2fa_code;
            VO_HMI_Status_Message := 'Gateway: Запрос охраны принят';
        E_Gateway_Command_Type.CMD_SET_TEMP: // Управление температурой
            IF (L_Process_Command.target_zone >= 1) AND (L_Process_Command.target_zone <= 32) THEN
                VO_Set_Temp_Req := TRUE;
                VO_Target_Zone := L_Process_Command.target_zone;
                VO_Target_Temp := L_Process_Command.target_value;
                VO_HMI_Status_Message := 'Gateway: Уставка температуры изменена';
            END_IF;
        E_Gateway_Command_Type.CMD_SET_VENT: // Управление вентиляцией
            // Пример: изменение скорости притока
            VO_Set_Vent_Req := TRUE;
            VO_Target_Vent_Speed := TO_BYTE(L_Process_Command.target_value);
            VO_HMI_Status_Message := 'Gateway: Уставка вентиляции изменена';
        E_Gateway_Command_Type.CMD_TELEGRAM_MSG: // Отправка сообщения в Telegram
            VO_Telegram_Msg := L_Process_Command.telegram_msg;
            VO_Send_Telegram := TRUE;
            VO_HMI_Status_Message := 'Gateway: Сообщение Telegram отправлено';
            VO_Sync_Time_Req := TRUE;
            VO_New_Time_MS := TO_UDINT(L_Process_Command.target_value);
            VO_HMI_Status_Message := 'Gateway: Время синхронизировано';
        END_CASE;
    END_IF;
ELSE
    VO_HMI_Status_Message := 'Gateway: Ошибка CRC команды';
END_IF;
END_IF;
// >>> BULK_SYNC_ANCHOR: FB_Gateway_Interface <<<

(* ---- FB_Heating_V2_Staging.st ---- *)
FUNCTION_BLOCK FB_Heating_V2_Staging
VAR_INPUT
    VI_Zone_ID : INT;
    VI_Enable : BOOL;
    VI_Target_Temp : REAL;
    VI_Valve_Position_Setpoint : REAL;
    VI_Pump_Enable : BOOL;
    VI_Is_Active : BOOL;
    VI_Room_Temp : REAL;
    VI_Supply_Temp : REAL;
    VI_Return_Temp : REAL;
    VI_Valve_Position_Actual : REAL;
    VI_Alarm_Active : BOOL;
END_VAR
VAR_OUTPUT
    VO_Command_Shadow : ST_Heating_Command_V2;
    VO_State_Shadow : ST_Heating_State_V2;
END_VAR

VO_Command_Shadow.Valve_Position_Setpoint := VI_Valve_Position_Setpoint;
VO_State_Shadow.Room_Temp := VI_Room_Temp;
VO_State_Shadow.Supply_Temp := VI_Supply_Temp;
END_FUNCTION_BLOCK

(* ---- FB_Maintenance_Access.st ---- *)
FUNCTION_BLOCK FB_Maintenance_Access
VAR_INPUT
    VI_System_Time : UDINT;
    VI_Activate    : BOOL;
    VI_Duration    : UDINT := 60; // мин
END_VAR
VAR_OUTPUT
    VO_Active      : BOOL;
    VO_Time_Left   : UDINT;
END_VAR
VAR
    L_Start_Time   : UDINT;
    L_elapsed      : UDINT;
END_VAR

IF VI_Activate AND NOT VO_Active THEN
    VO_Active := TRUE;
    L_Start_Time := VI_System_Time;
END_IF;

IF VO_Active THEN
    L_elapsed := (SEL(VI_System_Time >= L_Start_Time, VI_System_Time - L_Start_Time, (4294967295 - L_Start_Time) + VI_System_Time + 1)) / GVL_CONSTANTS.C_MS_IN_MINUTE;
    IF L_elapsed >= VI_Duration THEN
        VO_Active := FALSE;
    ELSE
        VO_Time_Left := VI_Duration - L_elapsed;
    END_IF;
END_IF;

(* ---- FB_Manual_Valve_Control.st ---- *)
FUNCTION_BLOCK FB_Manual_Valve_Control
VAR_INPUT
    VI_System_Time : UDINT;
    VI_Open_Req    : BOOL;
    VI_Duration    : UDINT := 5; // мин
END_VAR
VAR_OUTPUT
    VO_Open_Cmd    : BOOL;
    VO_Time_Left   : UDINT;
END_VAR
VAR
    L_Start_Time   : UDINT;
    L_Active       : BOOL;
    L_elapsed      : UDINT;
END_VAR

// Логика ручного управления клапаном с таймером автозакрытия
IF VI_Open_Req AND NOT L_Active THEN
    L_Active := TRUE;
    L_Start_Time := VI_System_Time;
    VO_Open_Cmd := TRUE;
END_IF;

IF L_Active THEN
    // Расчет оставшегося времени в минутах
    L_elapsed := (SEL(VI_System_Time >= L_Start_Time, VI_System_Time - L_Start_Time, (4294967295 - L_Start_Time) + VI_System_Time + 1)) / GVL_CONSTANTS.C_MS_IN_MINUTE;
    IF L_elapsed >= VI_Duration THEN
        L_Active := FALSE;
        VO_Open_Cmd := FALSE;
    ELSE
        VO_Time_Left := VI_Duration - L_elapsed;
    END_IF;
ELSE
    VO_Time_Left := 0;
END_IF;

(* ---- FB_Socket_Manager.st ---- *)
FUNCTION_BLOCK FB_Socket_Manager
// Менеджер управления розетками.
// Обеспечивает работу по сценариям, правилам и аварийное отключение (без локальных выключателей розеток).
VAR_INPUT
    VI_System_Time_MS : UDINT; // Системное время в миллисекундах
    VI_IsActivePLC : BOOL; // Флаг активности ПЛК (TRUE = ведущий)
    VI_Scenario : E_SCENARIO_TYPE; // Текущий глобальный сценарий
    VI_Fire_Alarm : BOOL; // Флаг пожарной тревоги
    VI_Flood_Alarm : BOOL; // Флаг тревоги протечки
    VI_Security_Armed : BOOL; // Состояние охраны (TRUE = включена)
END_VAR
VAR_IN_OUT
    VI_Manual_Override : ARRAY[1..GVL_CONSTANTS.C_MAX_SOCKETS] OF BOOL; // Ручное переопределение состояния (HMI)
    VI_Physical_Switches : ARRAY[1..GVL_CONSTANTS.C_MAX_SOCKETS] OF BOOL; // Legacy-вход: не используется в текущей концепции
    VI_Rule_Actions : ARRAY[1..GVL_CONSTANTS.C_MAX_RULES] OF ST_Rule_Action; // Действия от Rule Engine
    VI_IO_Modules_Online : ARRAY[1..GVL_CONSTANTS.C_MAX_MODULES] OF BOOL; // Статусы модулей ввода-вывода
END_VAR
VAR_OUTPUT
    VO_Socket_States : ARRAY[1..GVL_CONSTANTS.C_MAX_SOCKETS] OF BOOL; // Выходные состояния розеток
    VO_Internal_States : ARRAY[1..GVL_CONSTANTS.C_MAX_SOCKETS] OF BOOL; // Внутренние состояния для репликации
END_VAR
VAR
    // Socket V2 shadow (phase2)
    fbSocketV2Staging : FB_Socket_V2_Staging;
    L_Socket_V2_Command_Shadow : ST_Socket_Command_V2;
    L_Socket_V2_State_Shadow : ST_Socket_State_V2;
    L_Socket_V2_Shadow_Diff_Found : BOOL;
    L_Socket_V2_Switch_Enabled : BOOL;
    L_Socket_V2_Path_Ready : BOOL;
    L_Socket_Using_Legacy_Fallback : BOOL;
    L_i : INT;
    L_j : INT;
    L_Rule_State : BOOL;
    L_Rule_Active : BOOL;
    L_Internal_State : ARRAY[1..GVL_CONSTANTS.C_MAX_SOCKETS] OF BOOL;
    L_Manual_Trig : ARRAY[1..GVL_CONSTANTS.C_MAX_SOCKETS] OF R_TRIG;
END_VAR

IF NOT VI_IsActivePLC THEN RETURN; END_IF;

L_Socket_V2_Shadow_Diff_Found := FALSE;
L_Socket_V2_Switch_Enabled := TRUE;
L_Socket_V2_Path_Ready := FALSE;
L_Socket_Using_Legacy_Fallback := TRUE;

// Проверка связи с модулями ввода-вывода
FOR L_i := 1 TO GVL_CONSTANTS.C_MAX_MODULES DO
    IF NOT VI_IO_Modules_Online[L_i] THEN
        // Переход в безопасное состояние при потере связи (отключение всех розеток)
        FOR L_j := 1 TO GVL_CONSTANTS.C_MAX_SOCKETS DO
            VO_Socket_States[L_j] := FALSE;
        END_FOR;
        RETURN;
    END_IF;
END_FOR;

FOR L_i := 1 TO GVL_CONSTANTS.C_MAX_SOCKETS DO
    L_Rule_Active := FALSE;
    L_Rule_State := FALSE;

    L_Manual_Trig[L_i](CLK := VI_Manual_Override[L_i]);

    // Ручное переключение
    IF L_Manual_Trig[L_i].Q THEN
        L_Internal_State[L_i] := NOT L_Internal_State[L_i];
    END_IF;

    // Проверка правил для текущей розетки
    FOR L_j := 1 TO GVL_CONSTANTS.C_MAX_RULES DO
        IF VI_Rule_Actions[L_j].Active AND VI_Rule_Actions[L_j].Target_ID = L_i THEN
            IF VI_Rule_Actions[L_j].Action_Type = E_Rule_Action_Type.ACTION_SET_SOCKET THEN
                L_Rule_Active := TRUE;
                L_Rule_State := (VI_Rule_Actions[L_j].Value > 0.5);
                L_Internal_State[L_i] := L_Rule_State; // Синхронизация внутреннего состояния
            ELSIF VI_Rule_Actions[L_j].Action_Type = E_Rule_Action_Type.ACTION_TOGGLE_SOCKET AND VI_Rule_Actions[L_j].Triggered THEN
                L_Internal_State[L_i] := NOT L_Internal_State[L_i]; // Toggle
            END_IF;
        END_IF;
    END_FOR;

    // Аварийное отключение
    IF VI_Fire_Alarm OR VI_Flood_Alarm THEN
        // Розетки 1-4 неотключаемые (холодильник, сервер и т.д.)
        IF L_i > 4 THEN
            VO_Socket_States[L_i] := FALSE;
        ELSE
            // Критические розетки сохраняют свое текущее внутреннее состояние, а не форсируются в TRUE
            VO_Socket_States[L_i] := L_Internal_State[L_i];
        END_IF;
    ELSIF VI_Scenario = E_SCENARIO_TYPE.SCENARIO_AWAY OR VI_Security_Armed THEN
        // Master Off
        IF L_i > 4 THEN
            VO_Socket_States[L_i] := FALSE;
        ELSE
            // Неотключаемые розетки могут управляться вручную
            VO_Socket_States[L_i] := L_Internal_State[L_i];
        END_IF;
    ELSE
        // Нормальный режим: состояние определяется внутренним состоянием (ручным или правилом)
        IF L_Rule_Active THEN
            VO_Socket_States[L_i] := L_Rule_State;
        ELSE
            VO_Socket_States[L_i] := L_Internal_State[L_i];
        END_IF;
    END_IF;
END_FOR;

VO_Internal_States := L_Internal_State;

// ========================================
// Socket V2 shadow execution (phase2)
// ========================================
fbSocketV2Staging(
    VI_Socket_ID := 1,
    VI_Enable := TRUE,
    VI_Target_State := VO_Socket_States[1],
    VI_Manual_Override := VI_Manual_Override[1],
    VI_Safety_Lock := (VI_Fire_Alarm OR VI_Flood_Alarm),
    VI_Scenario_ID := TO_INT(VI_Scenario),

    VI_Is_On := VO_Socket_States[1],
    VI_Manual_Override_Active := VI_Manual_Override[1],
    VI_Safety_Blocked := (VI_Fire_Alarm OR VI_Flood_Alarm),
    VI_Alarm_Active := (VI_Fire_Alarm OR VI_Flood_Alarm),

    VO_Command_Shadow => L_Socket_V2_Command_Shadow,
    VO_State_Shadow => L_Socket_V2_State_Shadow
);

// ========================================
// Socket V2 shadow validation
// ========================================
IF VO_Socket_States[1] <> L_Socket_V2_Command_Shadow.Target_State THEN
    L_Socket_V2_Shadow_Diff_Found := TRUE;
END_IF;
IF VO_Socket_States[1] <> L_Socket_V2_State_Shadow.Is_On THEN
    L_Socket_V2_Shadow_Diff_Found := TRUE;
END_IF;
IF (VI_Fire_Alarm OR VI_Flood_Alarm) <> L_Socket_V2_State_Shadow.Safety_Blocked THEN
    L_Socket_V2_Shadow_Diff_Found := TRUE;
END_IF;

// Guarded Socket V2 enable
IF L_Socket_V2_Switch_Enabled THEN
    IF NOT L_Socket_V2_Shadow_Diff_Found THEN
        L_Socket_V2_Path_Ready := TRUE;
        L_Socket_Using_Legacy_Fallback := FALSE;
    ELSE
        L_Socket_V2_Path_Ready := FALSE;
        L_Socket_Using_Legacy_Fallback := TRUE;
    END_IF;
ELSE
    L_Socket_V2_Path_Ready := FALSE;
    L_Socket_Using_Legacy_Fallback := TRUE;
END_IF;

END_FUNCTION_BLOCK
// >>> BULK_SYNC_ANCHOR: FB_Socket_Manager <<<

(* ---- FB_System_Timer.st ---- *)
// ==============================================================================
// Блок таймера, привязанный к системному времени (System Timer)
// Назначение:
// - Замена стандартного TON для обеспечения точной выдержки времени,
//   независимой от времени цикла ПЛК, с использованием единого системного времени.
// ==============================================================================
FUNCTION_BLOCK FB_System_Timer
VAR_INPUT
    IN : BOOL; // Вход запуска таймера
    PT : TIME; // Заданное время
    VI_System_Time_MS : UDINT; // Системное время (мс)
END_VAR
VAR_OUTPUT
    Q : BOOL; // Выход: таймер сработал
    ET : TIME; // Прошедшее время
END_VAR
VAR
    L_Start_Time : UDINT;
    L_Running : BOOL;
END_VAR

IF IN THEN
    IF NOT L_Running THEN
        L_Start_Time := VI_System_Time_MS;
        L_Running := TRUE;
        ET := T#0s;
        Q := FALSE;
    ELSE
        // Обработка переполнения UDINT (примерно 49 дней)
        ET := TO_TIME((SEL(VI_System_Time_MS >= L_Start_Time, VI_System_Time_MS - L_Start_Time, (4294967295 - L_Start_Time) + VI_System_Time_MS + 1)));

        IF ET >= PT THEN
            Q := TRUE;
            ET := PT;
        ELSE
            Q := FALSE;
        END_IF;
    END_IF;
ELSE
    L_Running := FALSE;
    ET := T#0s;
    Q := FALSE;
END_IF;
// >>> BULK_SYNC_ANCHOR: FB_System_Timer <<<

(* ---- FB_Water_Leakage_Manager.st ---- *)
FUNCTION_BLOCK FB_Water_Leakage_Manager
VAR_INPUT
    VI_System_Time_MS : UDINT;
    VI_IsActivePLC    : BOOL;
    VI_Config         : ST_Flood_Global_Config;
END_VAR

VAR_IN_OUT
    VI_Sensors : ARRAY[1..GVL_CONSTANTS.C_MAX_FLOOD_SENSORS] OF BOOL;
END_VAR

VAR_OUTPUT
    VO_Close_Valve_35 : BOOL;
    VO_Close_Valve_36 : BOOL;
    VO_Status_Msg     : STRING(200);

    // Health signals
    VO_Leak_Detected      : BOOL;
    VO_Leak_Warning_Level : BOOL;
END_VAR

VAR
    L_i             : INT;
    L_Sensor_Timers : ARRAY[1..GVL_CONSTANTS.C_MAX_FLOOD_SENSORS] OF FB_System_Timer;
    L_Any_Leak      : BOOL;
    L_Any_Warning   : BOOL;
END_VAR

IF NOT VI_IsActivePLC THEN RETURN; END_IF;

L_Any_Leak := FALSE;
L_Any_Warning := FALSE;

FOR L_i := 1 TO GVL_CONSTANTS.C_MAX_FLOOD_SENSORS DO
    L_Sensor_Timers[L_i](
        IN := VI_Sensors[L_i],
        PT := TO_TIME(VI_Config.min_duration_ms + VI_Config.warning_duration_ms),
        VI_System_Time_MS := VI_System_Time_MS
    );

    IF L_Sensor_Timers[L_i].ET >= TO_TIME(VI_Config.min_duration_ms) THEN
        L_Any_Warning := TRUE;

        IF L_Sensor_Timers[L_i].Q THEN
            L_Any_Leak := TRUE;

            IF VI_Config.sensor_to_valve_map[L_i] = 1 THEN
                VO_Close_Valve_35 := TRUE;
            ELSIF VI_Config.sensor_to_valve_map[L_i] = 2 THEN
                VO_Close_Valve_36 := TRUE;
            END_IF;
        END_IF;
    END_IF;
END_FOR;

// Health signals
VO_Leak_Detected := L_Any_Leak;
VO_Leak_Warning_Level := L_Any_Warning;

// Status
IF L_Any_Leak THEN
    VO_Status_Msg := 'АВАРИЯ: ПРОТЕЧКА ВОДЫ. КЛАПАНЫ ЗАКРЫТЫ.';
ELSIF L_Any_Warning THEN
    VO_Status_Msg := 'ПРЕДУПРЕЖДЕНИЕ: ОБНАРУЖЕНА ВОДА.';
ELSE
    VO_Status_Msg := 'Система контроля протечек в норме';
    VO_Close_Valve_35 := FALSE;
    VO_Close_Valve_36 := FALSE;
END_IF;
// >>> BULK_SYNC_ANCHOR: FB_Water_Leakage_Manager <<<

(* ---- FB_Water_Valve_Controller.st ---- *)
FUNCTION_BLOCK FB_Water_Valve_Controller IMPLEMENTS IValveController
VAR_INPUT
    VI_System_Time : UDINT;
    VI_IsActivePLC : BOOL;
    VI_Flood_Alarm : BOOL;
END_VAR
VAR_OUTPUT
    VO_Valve_Closed : BOOL;
    VO_Status_Msg   : STRING(200);
END_VAR

IF VI_Flood_Alarm AND VI_IsActivePLC THEN
    VO_Valve_Closed := TRUE;
    VO_Status_Msg := 'КЛАПАН ЗАКРЫТ ПО ПРОТЕЧКЕ';
END_IF;

METHOD OpenValve : BOOL
VAR_INPUT
    VI_Operator_ID : STRING(10);
    VI_Force : BOOL;
END_VAR
IF VI_IsActivePLC OR VI_Force THEN
    VO_Valve_Closed := FALSE;
    OpenValve := TRUE;
END_IF;
END_METHOD

METHOD CloseValve : BOOL
VAR_INPUT
    VI_Operator_ID : STRING(10);
    VI_Force : BOOL;
END_VAR
VO_Valve_Closed := TRUE;
CloseValve := TRUE;
END_METHOD

METHOD GetStatus : BYTE
GetStatus := TO_BYTE(SEL(VO_Valve_Closed, 0, 1));
END_METHOD

(* ---- PRG_Heating.st ---- *)
PROGRAM PRG_Heating
VAR
    fbHeatingManager : FB_Heating_System_Manager;
    fbDHWManager : FB_DHW_Manager;
    L_i : INT;
    L_Zone_Valves_8 : ARRAY[1..8] OF BOOL;
    L_Boiler_Modulation_REAL : ARRAY[1..GVL_CONSTANTS.C_MAX_BOILERS] OF REAL;
END_VAR

FOR L_i := 1 TO GVL_CONSTANTS.C_MAX_BOILERS DO
    L_Boiler_Modulation_REAL[L_i] := TO_REAL(GVL_IO.AI_Boiler_Modulation[L_i]);
END_FOR;

// 9. Управление климатом (Отопление)
fbHeatingManager(
    VI_System_Time_MS := GVL_STATUS.G_System_Time_MS,
    VI_Current_TOD := GVL_STATUS.G_Current_TOD,
    VI_IsActivePLC := GVL_STATUS.G_Is_Active_PLC,
    VI_Outdoor_Temp := GVL_STATE.G_Outdoor_Temp,
    VI_Floor_Temps := GVL_STATE.G_Floor_Temps,
    VI_Room_Temps := GVL_STATE.G_Room_Temps,
    VI_Config := GVL_CONFIG.G_Heating_Config,
    VI_Zone_Configs := GVL_CONFIG.G_HMI_FloorHeating_Configs,
    VI_Tariff := GVL_CONFIG.G_HMI_Tariff_Settings,
    VI_Current_Hour := TO_UINT(GVL_STATUS.G_Time_Of_Day_MS / GVL_CONSTANTS.C_MS_IN_HOUR),
    VI_Manifold_Pressures := GVL_STATE.G_Manifold_Pressures,
    VI_Manifold_Currents := GVL_STATE.G_Manifold_Currents,
    VI_Manifold_Temps_Supply := GVL_STATE.G_Manifold_T_Supply,
    VI_Manifold_Temps_Return := GVL_STATE.G_Manifold_T_Return,
    VI_Boiler_Flame_Status := GVL_STATE.G_Boiler_Flame,
    VI_Boiler_Error_Status := GVL_STATE.G_Boiler_Error,
    VI_Boiler_OT_Online := GVL_STATE.G_Boiler_OT_Online,
    VI_Boiler_Modulation := L_Boiler_Modulation_REAL,
    VI_Rule_Actions := GVL_STATE.G_Rule_Actions,
    VI_Boiler_Stop := GVL_COMMAND.G_Boiler_Stop,
    VI_IO_Modules_Online := GVL_STATUS.G_IO_Modules_Online,
    VI_DHW_Heating_Demand := fbDHWManager.VO_Heating_Pump,
    VI_DHW_Target_Temp := GVL_CONFIG.G_DHW_Config.Target_Temp,
    VI_Current_Scenario := GVL_STATUS.G_Current_Scenario,
    VI_System_Mode := GVL_STATE.G_System_Mode,
    VI_Emergency_Stop := GVL_STATE.G_Safety_Emergency_Stop,
    VI_Gas_Safety_Stop := GVL_STATE.G_Safety_Gas_Latched,
    VI_Scenario_Configs := GVL_CONFIG.G_HMI_Scenario_Configs,
    VI_Manifold_End_Switches := GVL_STATE.G_Manifold_End_Switches,
    VI_Valve_Test_Config := GVL_CONFIG.G_Valve_Test_Config,
    VO_Manifold_Valves => GVL_STATE.G_Manifold_Valves,
    VO_Manifold_Pumps => GVL_STATE.G_Manifold_Pumps,
    VO_Zone_Valves => L_Zone_Valves_8,
    VO_Boiler_OT_Enable => GVL_STATE.G_Boiler_OT_Enable,
    VO_Boiler_OT_Setpoint => GVL_STATE.G_Boiler_OT_Setpoint,
    VO_Backup_Circulation_Pump => GVL_STATE.G_Backup_Circulation_Pump,
    VO_Electric_Heater_Enable => GVL_STATE.G_Electric_Heater_Enable,
    VO_Freeze_Risk_Status => GVL_STATE.G_Safety_Freeze_Risk,
    VO_Status => GVL_STATUS.G_Manifold_Status,
    VO_Boiler_Status => GVL_STATUS.G_Boiler_Status
);

// 12. Управление ГВС
fbDHWManager(
    VI_System_Time_MS := GVL_STATUS.G_System_Time_MS,
    VI_Current_TOD := GVL_STATUS.G_Current_TOD,
    VI_IsActivePLC := GVL_STATUS.G_Is_Active_PLC,
    VI_Temp := GVL_STATE.G_DHW_Temp,
    VI_Pressure := GVL_STATE.G_DHW_Pressure,
    VI_Config := GVL_CONFIG.G_DHW_Config,
    VI_Current_Day_Of_Week := GVL_STATUS.G_Current_Day,
    VI_IO_Modules_Online := GVL_STATUS.G_IO_Modules_Online,
    VI_Reset_Errors := GVL_COMMAND.G_Reset_Errors,
    VI_Emergency_Stop := GVL_STATE.G_Safety_Emergency_Stop,
    VO_Heating_Pump => GVL_STATE.G_DHW_Heating_Pump,
    VO_Circ_Pump => GVL_STATE.G_DHW_Circ_Pump,
    VO_Status => GVL_STATUS.G_DHW_Status
);

// Integrated freeze-hardware diagnostics and maintenance gating
GVL_STATUS.G_Diagnostics.Backup_Pump_Out_Of_Service := NOT GVL_CONFIG.G_Backup_Circulation_Pump_In_Service;
GVL_STATUS.G_Diagnostics.Electric_Heater_Out_Of_Service := NOT GVL_CONFIG.G_Electric_Heater_In_Service;
IF NOT GVL_CONFIG.G_Backup_Circulation_Pump_In_Service THEN
    GVL_STATE.G_Backup_Circulation_Pump := FALSE;
END_IF;
IF NOT GVL_CONFIG.G_Electric_Heater_In_Service THEN
    GVL_STATE.G_Electric_Heater_Enable := FALSE;
END_IF;

GVL_STATE.G_Freeze_Hardware_Degraded := GVL_STATUS.G_Diagnostics.Backup_Pump_Fault OR GVL_STATUS.G_Diagnostics.Electric_Heater_Fault;
GVL_STATE.G_Freeze_Hardware_Failed := GVL_STATUS.G_Diagnostics.Backup_Pump_Fault AND GVL_STATUS.G_Diagnostics.Electric_Heater_Fault;

IF GVL_STATE.G_Freeze_Hardware_Failed THEN
    GVL_STATE.G_Backup_Circulation_Pump := FALSE;
    GVL_STATE.G_Electric_Heater_Enable := FALSE;
    GVL_STATE.G_Safety_Freeze_Risk := TRUE;
END_IF;

FOR L_i := 1 TO GVL_CONSTANTS.C_MAX_MANIFOLDS DO
    GVL_STATUS.G_Diagnostics.Manifold_Pump_Out_Of_Service[L_i] := NOT GVL_CONFIG.G_Manifold_Pump_In_Service[L_i];
    IF NOT GVL_CONFIG.G_Manifold_Pump_In_Service[L_i] THEN
        GVL_STATE.G_Manifold_Pumps[L_i] := FALSE;
    END_IF;
END_FOR;
GVL_STATUS.G_Diagnostics.DHW_Heating_Pump_Out_Of_Service := NOT GVL_CONFIG.G_DHW_Heating_Pump_In_Service;
IF NOT GVL_CONFIG.G_DHW_Heating_Pump_In_Service THEN
    GVL_STATE.G_DHW_Heating_Pump := FALSE;
END_IF;
GVL_STATUS.G_Diagnostics.DHW_Circ_Pump_Out_Of_Service := NOT GVL_CONFIG.G_DHW_Circ_Pump_In_Service;
IF NOT GVL_CONFIG.G_DHW_Circ_Pump_In_Service THEN
    GVL_STATE.G_DHW_Circ_Pump := FALSE;
END_IF;
// >>> BULK_SYNC_ANCHOR: PRG_Heating <<<

// HEATING ADAPTER COPY OUT
FOR L_i := 1 TO 8 DO
    GVL_STATE.G_Zone_Valves[L_i] := L_Zone_Valves_8[L_i];
END_FOR;

(* ---- PRG_System.st ---- *)
PROGRAM PRG_System
VAR
    L_i : INT;
    L_Motion_Sensors_16 : ARRAY[1..16] OF BOOL;
    // --- ADAPTER LAYER ---
    L_Zone_Valves_8 : ARRAY[1..8] OF BOOL;
    L_Lighting_32   : ARRAY[1..32] OF BYTE;
    L_Lighting_Bool_32 : ARRAY[1..32] OF BOOL;
    L_FloorTemps_8  : ARRAY[1..8] OF REAL;
    fbCoreKernelObserver : FB_CoreKernel_Live_Observer;
    fbSystemHealth : FB_System_Health;
    fbRedundancy : FB_Redundancy_Manager;
    fbGateway : FB_Gateway_Interface;
    fbScenarioManager : FB_Scenario_Manager;
    fbSimulationManager : FB_Simulation_Manager;
    fbRuleEngine : FB_Rule_Engine;
    fbNVRAMManager : FB_NVRAM_Manager;
    fbBlackBox : FB_BlackBox_Recorder;
    fbAstroTimer : FB_Astro_Timer;
    fbAlarmManager : FB_Alarm_Manager;
    fbHistoryManager : FB_History_Manager;
    fbSafety : FB_Safety_Manager;
    fbStateManager : FB_State_Manager;
    fbWatchdog : FB_Watchdog;
    fbHMIInterface : FB_HMI_Interface;
    fbFaultLogger : FB_Fault_Logger;

    L_Time_Diff : UDINT;
    L_Local_State : ST_System_State_Snapshot;
    L_Remote_State : ST_System_State_Snapshot;
    L_Config_Loaded : BOOL;
    L_NVRAM_Cmd : BYTE;
    L_NVRAM_Offset : UDINT;
    L_NVRAM_Done : BOOL;
    L_NVRAM_Err : BOOL;
    L_NVRAM_ErrID : UDINT;
    L_BB_Record : ST_BlackBox_Record;
    L_BB_Freeze : BOOL;
    L_Scenario_Idx : INT;
        L_Last_Operator_Blocked : BOOL;
    L_Last_DHW_Heating_In_Service : BOOL;
    L_Last_DHW_Circ_In_Service : BOOL;
    L_Dangerous_Action_Armed : BOOL;
    L_Dangerous_Action_Deadline_MS : UDINT;
    L_Last_System_Mode : E_System_Operating_Mode;
    L_Last_First_Fault_Type : INT;
    L_Last_First_Fault_Source : INT;
    L_Last_Root_Cause : E_System_Root_Cause;
    L_History_Event : ST_History_Record;
    L_History_Write_Event : BOOL;
    L_Last_Operator_Journal_Seq : UDINT;
    L_Last_Event_Code : UDINT;
    L_Last_Event_Value : REAL;
    L_Last_Event_Time_MS : UDINT;
    L_Gateway_Writes_Allowed : BOOL;
END_VAR

// 0. Инициализация RETAIN переменных при первом запуске
IF NOT GVL_Retain.G_Initialized THEN
    FOR L_i := 0 TO GVL_CONSTANTS.C_MAX_PRESENCE_HISTORY - 1 DO
        GVL_Retain.G_Presence_History[L_i] := 0;
    END_FOR;

    GVL_Retain.G_History_Write_Idx := 1;
    GVL_Retain.G_History_Total_Events := 0;

    FOR L_i := 1 TO GVL_CONSTANTS.C_MAX_BOILERS DO
        GVL_Retain.G_Boiler_Accumulated_MS[L_i] := 0;
        GVL_Retain.G_Boiler_Work_Seconds[L_i] := 0;
    END_FOR;

    FOR L_i := 1 TO GVL_CONSTANTS.C_MAX_MANIFOLDS DO
        GVL_Retain.G_Valve_Test_Results[L_i] := FALSE;
    END_FOR;

    L_Local_State.Version := 0;
    L_Remote_State.Version := 0;

    GVL_Retain.G_Initialized := TRUE;
END_IF;

// 1. Обновление системного времени
GVL_STATUS.G_System_Time_MS := TIME_TO_UDINT(TIME());
L_Time_Diff := (SEL(GVL_STATUS.G_System_Time_MS >= GVL_STATUS.G_Last_System_Time_MS, GVL_STATUS.G_System_Time_MS - GVL_STATUS.G_Last_System_Time_MS, (4294967295 - GVL_STATUS.G_Last_System_Time_MS) + GVL_STATUS.G_System_Time_MS + 1));
GVL_STATUS.G_Time_Of_Day_MS := (GVL_STATUS.G_Time_Of_Day_MS + L_Time_Diff) MOD 86400000;

IF GVL_STATUS.G_Time_Of_Day_MS < L_Time_Diff THEN
    GVL_STATUS.G_Current_Day := (GVL_STATUS.G_Current_Day MOD 7) + 1;
    GVL_STATUS.G_Day_Of_Year := (GVL_STATUS.G_Day_Of_Year MOD 365) + 1;
END_IF;

GVL_STATUS.G_Last_System_Time_MS := GVL_STATUS.G_System_Time_MS;
GVL_STATUS.G_Current_TOD := UDINT_TO_TOD(GVL_STATUS.G_Time_Of_Day_MS);

// Формирование локального состояния для репликации
L_Local_State.System_Time_MS := GVL_STATUS.G_System_Time_MS;
L_Local_State.Current_Scenario := GVL_STATUS.G_Current_Scenario;
L_Local_State.Security_Armed := GVL_ALARM.G_Security_Armed;
L_Local_State.Active_Alarms := GVL_ALARM.G_Active_Alarm_Count;
L_Local_State.Zone_Valves := GVL_STATE.G_Zone_Valves;
L_Local_State.Manifold_Pumps := GVL_STATE.G_Manifold_Pumps;
L_Local_State.Lighting_States := GVL_STATE.G_Lighting_Levels;
L_Local_State.Blinds_Positions := GVL_STATE.G_Blinds_Positions;
L_Local_State.Socket_States := GVL_STATE.G_Socket_States;
L_Local_State.Gas_Valve_Closed := GVL_COMMAND.G_Gas_Valve_Close;
L_Local_State.Water_Valves_Closed := GVL_COMMAND.G_Close_Valve_36;
L_Local_State.Version := L_Local_State.Version + 1;

// 2. Определение роли ПЛК (Active/Standby)
fbRedundancy(
    VI_System_Time_MS := GVL_STATUS.G_System_Time_MS,
    VI_Local_PLC_ID := GVL_STATUS.G_PLC_ID,
    VI_Remote_Pulse := GVL_IO.DI_Partner_Pulse,
    VI_Remote_Is_Active := GVL_IO.DI_Partner_Active,
    VI_Gateway_Ping_OK := GVL_GATEWAY.G_Gateway_Ping_OK,
    VI_Local_State := L_Local_State,
    VI_Remote_State := L_Remote_State
);
GVL_STATUS.G_Is_Active_PLC := (fbRedundancy.VO_Local_Role = E_PLC_ROLE.ROLE_ACTIVE);
GVL_IO.DO_Heartbeat_Pulse := fbRedundancy.VO_Local_Pulse;
GVL_IO.DO_Active_Status := GVL_STATUS.G_Is_Active_PLC;

// 3. Синхронизация состояния (применение полученного состояния)
IF fbRedundancy.VO_State_Updated THEN
    GVL_STATUS.G_Current_Scenario := fbRedundancy.VO_Synced_State.Current_Scenario;
    GVL_ALARM.G_Security_Armed := fbRedundancy.VO_Synced_State.Security_Armed;
    GVL_STATE.G_Zone_Valves := fbRedundancy.VO_Synced_State.Zone_Valves;
    GVL_STATE.G_Manifold_Pumps := fbRedundancy.VO_Synced_State.Manifold_Pumps;
    GVL_STATE.G_Lighting_Levels := fbRedundancy.VO_Synced_State.Lighting_States;
    GVL_STATE.G_Blinds_Positions := fbRedundancy.VO_Synced_State.Blinds_Positions;
    GVL_STATE.G_Socket_States := fbRedundancy.VO_Synced_State.Socket_States;
    GVL_COMMAND.G_Gas_Valve_Close := fbRedundancy.VO_Synced_State.Gas_Valve_Closed;
    GVL_COMMAND.G_Close_Valve_36 := fbRedundancy.VO_Synced_State.Water_Valves_Closed;
    L_Local_State.Version := fbRedundancy.VO_Synced_State.Version;
END_IF;

fbSafety(
    VI_Gas_Alarm := GVL_STATE.G_Safety_Gas_Alarm,
    VI_Leak_Alarm := GVL_STATE.G_Safety_Leak_Alarm,
    VI_Smoke_Alarm := GVL_STATE.G_Safety_Smoke_Alarm,
    VI_Reset := GVL_COMMAND.G_Reset_Errors,
    VO_Gas_Latched => GVL_STATE.G_Safety_Gas_Latched,
    VO_Leak_Latched => GVL_STATE.G_Safety_Leak_Latched,
    VO_Smoke_Latched => GVL_STATE.G_Safety_Smoke_Latched,
    VO_Emergency_Stop => GVL_STATE.G_Safety_Emergency_Stop
);

// 3.4. Агрегация состояния anti-freeze hardware
GVL_STATE.G_Freeze_Hardware_Degraded := GVL_STATUS.G_Diagnostics.Backup_Pump_Fault OR GVL_STATUS.G_Diagnostics.Electric_Heater_Fault;
GVL_STATE.G_Freeze_Hardware_Failed := GVL_STATUS.G_Diagnostics.Backup_Pump_Fault AND GVL_STATUS.G_Diagnostics.Electric_Heater_Fault;

// 3.6. Health manager: новая интеграция safety + diagnostics + watchdog
fbWatchdog(
    VI_System_Time_MS := GVL_STATUS.G_System_Time_MS
);

fbSystemHealth(
    VI_Smoke_Detected := GVL_HEALTH_BRIDGE.G_Smoke_Detected OR GVL_STATE.G_Safety_Smoke_Latched,
    VI_Gas_Detected := GVL_HEALTH_BRIDGE.G_Gas_Detected OR GVL_STATE.G_Safety_Gas_Latched,
    VI_CO_Warning_Level := GVL_HEALTH_BRIDGE.G_CO_Warning_Level,
    VI_CO_Alarm_Level := GVL_HEALTH_BRIDGE.G_CO_Alarm_Level,
    VI_Leak_Detected := GVL_HEALTH_BRIDGE.G_Leak_Detected OR GVL_STATE.G_Safety_Leak_Latched,
    VI_Sensor_Fault := GVL_STATE.G_Heating_Sensor_Fault OR GVL_STATE.G_DHW_Sensor_Fault,
    VI_IO_Offline := GVL_STATE.G_Heating_IO_Fault OR GVL_STATE.G_DHW_IO_Fault OR GVL_STATE.G_Ventilation_IO_Fault OR GVL_STATE.G_Lighting_IO_Fault,
    VI_Comm_Fault := GVL_STATE.G_Access_Comm_Fault,
    VI_Watchdog_Fault := fbWatchdog.VO_Watchdog_Fault,
    VI_Subsystem_Fault := GVL_STATE.G_Heating_Subsystem_Degraded OR GVL_STATE.G_DHW_Subsystem_Degraded OR GVL_STATE.G_Ventilation_Subsystem_Degraded
);

// 3.6. State manager: агрегированная логика режима работы
fbStateManager(
    VI_System_Severity := fbSystemHealth.VO_System_Severity,
    VI_Root_Cause := fbSystemHealth.VO_Root_Cause,
    VI_Freeze_Risk := GVL_STATE.G_Safety_Freeze_Risk
);

fbHMIInterface(
    VI_Severity := fbSystemHealth.VO_System_Severity,
    VI_RootCause := fbSystemHealth.VO_Root_Cause,
    VI_Status_Msg := fbStateManager.VO_Status_Msg
);

fbFaultLogger(
    VI_Severity := fbSystemHealth.VO_System_Severity,
    VI_RootCause := fbSystemHealth.VO_Root_Cause,
    VI_Time_MS := GVL_STATUS.G_System_Time_MS
);

// publish integrated outputs
GVL_STATUS.G_System_Mode_Msg := fbStateManager.VO_Status_Msg;

// === DIAGNOSTIC FLAGS (export) ===
GVL_STATUS.G_Diagnostics.Sensor_Fault :=
    GVL_STATE.G_Heating_Sensor_Fault OR
    GVL_STATE.G_DHW_Sensor_Fault;

GVL_STATUS.G_Diagnostics.IO_Offline :=
    GVL_STATE.G_Heating_IO_Fault OR
    GVL_STATE.G_DHW_IO_Fault OR
    GVL_STATE.G_Ventilation_IO_Fault OR
    GVL_STATE.G_Lighting_IO_Fault;

GVL_STATUS.G_Diagnostics.Subsystem_Degraded :=
    GVL_STATE.G_Heating_Subsystem_Degraded OR
    GVL_STATE.G_DHW_Subsystem_Degraded OR
    GVL_STATE.G_Ventilation_Subsystem_Degraded;

GVL_GATEWAY.G_Gateway_HMI_Status_Message := fbHMIInterface.VO_HMI_Status_Text;
IF fbFaultLogger.VO_Last_Event_Text <> '' THEN
    GVL_HEALTH_BRIDGE.G_Last_Fault_Event_Text := fbFaultLogger.VO_Last_Event_Text;
END_IF;

// 3.7. Применение вычисленного режима системы
GVL_STATE.G_System_Mode := fbStateManager.VO_System_Mode;

CASE GVL_STATE.G_System_Mode OF
    E_System_Operating_Mode.MODE_SAFE_STOP:
        GVL_STATE.G_System_Mode_Text := 'SAFE_STOP';

    E_System_Operating_Mode.MODE_FREEZE_PROTECTION:
        GVL_STATE.G_System_Mode_Text := 'FREEZE_PROTECTION';

    E_System_Operating_Mode.MODE_DEGRADED:
        GVL_STATE.G_System_Mode_Text := 'DEGRADED';

    ELSE
        GVL_STATE.G_System_Mode_Text := 'NORMAL';
END_CASE;

CASE fbSystemHealth.VO_Root_Cause OF
    E_System_Root_Cause.ROOT_FIRE:
        GVL_STATUS.G_System_Mode_Cause := 'Пожар/дым';
    E_System_Root_Cause.ROOT_GAS_LEAK:
        GVL_STATUS.G_System_Mode_Cause := 'Утечка газа';
    E_System_Root_Cause.ROOT_CO_CRITICAL:
        GVL_STATUS.G_System_Mode_Cause := 'Критический CO';
    E_System_Root_Cause.ROOT_CO_WARNING:
        GVL_STATUS.G_System_Mode_Cause := 'Повышенный CO';
    E_System_Root_Cause.ROOT_WATER_LEAK:
        GVL_STATUS.G_System_Mode_Cause := 'Протечка воды';
    E_System_Root_Cause.ROOT_WATCHDOG_FAULT:
        GVL_STATUS.G_System_Mode_Cause := 'Ошибка watchdog';
    E_System_Root_Cause.ROOT_IO_OFFLINE:
        GVL_STATUS.G_System_Mode_Cause := 'Недоступен модуль IO';
    E_System_Root_Cause.ROOT_COMM_FAULT:
        GVL_STATUS.G_System_Mode_Cause := 'Ошибка связи';
    E_System_Root_Cause.ROOT_SENSOR_FAULT:
        GVL_STATUS.G_System_Mode_Cause := 'Ошибка датчика';
    E_System_Root_Cause.ROOT_SUBSYSTEM_FAULT:
        GVL_STATUS.G_System_Mode_Cause := 'Ошибка подсистемы';
    ELSE
        GVL_STATUS.G_System_Mode_Cause := 'Аварийные режимы отсутствуют';
END_CASE;

// final status text comes from State_Manager
GVL_STATUS.G_System_Mode_Msg := fbStateManager.VO_Status_Msg;

// 3.6a. Расчёт направленной эвакуации
FOR L_i := 1 TO 32 DO
    GVL_STATE.G_Evac_Guidance[L_i] := 0;

    IF GVL_STATE.G_Evac_Hazard_Zone[L_i] THEN
        GVL_STATE.G_Evac_Guidance[L_i] := -1;
    END_IF;

    IF GVL_CONFIG.G_Evac_Exit_Zones[L_i] AND NOT GVL_STATE.G_Evac_Hazard_Zone[L_i] THEN
        GVL_STATE.G_Evac_Guidance[L_i] := 1;
    END_IF;
END_FOR;

// 3.5a. Вычисление человекочитаемых имён зон эвакуации для HMI
GVL_STATUS.G_Evac_Target_Zone_Name := '';
GVL_STATUS.G_Evac_Hazard_Zone_Name := '';

FOR L_i := 1 TO 32 DO
    IF (GVL_STATUS.G_Evac_Hazard_Zone_Name = '') AND GVL_STATE.G_Evac_Hazard_Zone[L_i] THEN
        GVL_STATUS.G_Evac_Hazard_Zone_Name := GVL_CONFIG.G_Evac_Zone_Names[L_i];
        IF GVL_STATUS.G_Evac_Hazard_Zone_Name = '' THEN
            GVL_STATUS.G_Evac_Hazard_Zone_Name := CONCAT('Zone ', INT_TO_STRING(L_i));
        END_IF;
    END_IF;

    IF (GVL_STATUS.G_Evac_Target_Zone_Name = '') AND (GVL_STATE.G_Evac_Guidance[L_i] = 1) THEN
        GVL_STATUS.G_Evac_Target_Zone_Name := GVL_CONFIG.G_Evac_Zone_Names[L_i];
        IF GVL_STATUS.G_Evac_Target_Zone_Name = '' THEN
            GVL_STATUS.G_Evac_Target_Zone_Name := CONCAT('Zone ', INT_TO_STRING(L_i));
        END_IF;
    END_IF;
END_FOR;

// 3.6. Активация световой эвакуации
IF GVL_STATE.G_System_Mode = E_System_Operating_Mode.MODE_SAFE_STOP AND GVL_STATE.G_Safety_Smoke_Latched THEN
    GVL_STATE.G_Evacuation_Lighting_Active := TRUE;
ELSE
    GVL_STATE.G_Evacuation_Lighting_Active := FALSE;
END_IF;

// 4. Астрономический таймер
fbAstroTimer(
    VI_System_Time_MS := GVL_STATUS.G_System_Time_MS,
    VI_Latitude := 55.75,
    VI_Longitude := 37.61,
    VI_Day_Of_Year := GVL_STATUS.G_Day_Of_Year,
    VO_Is_Night => GVL_STATUS.G_Is_Night
);

// 5. Управление сценариями
fbScenarioManager(
    VI_System_Time_MS := GVL_STATUS.G_System_Time_MS,
    VI_Activate_Request := GVL_COMMAND.G_Scenario_Request,
    VI_IsActivePLC := GVL_STATUS.G_Is_Active_PLC,
    VI_System_Mode := GVL_STATE.G_System_Mode,
    VO_Current_Scenario => GVL_STATUS.G_Current_Scenario
);

// Синхронизируем request с фактически активным сценарием
GVL_COMMAND.G_Scenario_Request := GVL_STATUS.G_Current_Scenario;

L_Scenario_Idx := TO_INT(GVL_STATUS.G_Current_Scenario);
IF L_Scenario_Idx < 1 OR L_Scenario_Idx > 6 THEN
    L_Scenario_Idx := 1;
END_IF;

// 6. Симуляция присутствия
fbSimulationManager(
    VI_System_Time_MS := GVL_STATUS.G_System_Time_MS,
    VI_IsActivePLC := GVL_STATUS.G_Is_Active_PLC AND (GVL_STATE.G_System_Mode = E_System_Operating_Mode.MODE_NORMAL),
    VI_Scenario := GVL_STATUS.G_Current_Scenario,
    VI_Config := GVL_CONFIG.G_HMI_Scenario_Configs[L_Scenario_Idx],
    VO_Sim_Lights => GVL_STATE.G_Sim_Lights,
    VO_Sim_Active => GVL_STATUS.G_Sim_Active
);

// 6.5. Пользовательские правила (Rule Engine)
fbRuleEngine(
    VI_System_Time_MS := GVL_STATUS.G_System_Time_MS,
    VI_IsActivePLC := GVL_STATUS.G_Is_Active_PLC,
    VI_Rules := GVL_CONFIG.G_HMI_User_Rules,
    VI_Indoor_Temps := GVL_STATE.G_Room_Temps,
    VI_Floor_Temps := L_FloorTemps_8,
    VI_Humidities := GVL_STATE.G_Room_Hum,
    VI_CO2_Levels := GVL_STATE.G_Room_CO2,
    VI_Motion_Sensors := L_Motion_Sensors_16,
    VI_Door_Sensors := GVL_STATE.G_Door_Sensors,
    VI_Window_Sensors := GVL_STATE.G_Window_Sensors,
    VI_Water_Sensors := GVL_STATE.G_Water_Sensors,
    VI_Smoke_Sensors := GVL_STATE.G_Smoke_Sensors,
    VI_Methane_Sensors := GVL_STATE.G_Methane_Sensors,
    VI_CO_Sensors := GVL_STATE.G_CO_Sensors,
    VI_Security_Armed := GVL_ALARM.G_Security_Armed,
    VI_Current_Time := GVL_STATUS.G_Current_TOD,
    VI_Day_Of_Week := TO_INT(GVL_STATUS.G_Current_Day),
    VO_Actions => GVL_STATE.G_Rule_Actions
);

FOR L_i := 1 TO GVL_CONSTANTS.C_MAX_RULES DO
    IF GVL_STATE.G_Rule_Actions[L_i].Active AND GVL_STATE.G_Rule_Actions[L_i].Action_Type = E_Rule_Action_Type.ACTION_ACTIVATE_SCENARIO THEN
        GVL_COMMAND.G_Scenario_Request := TO_BYTE(GVL_STATE.G_Rule_Actions[L_i].Value);
    END_IF;
END_FOR;

// 8.5 Менеджер тревог (Сбор всех аварий)
fbAlarmManager(
    VI_System_Time_MS := GVL_STATUS.G_System_Time_MS,
    VI_IsActivePLC := GVL_STATUS.G_Is_Active_PLC,
    VI_Gas_Alarm := GVL_ALARM.G_Gas_Alarm_Active,
    VI_Fire_Alarm := GVL_ALARM.G_Fire_Alarm_Active,
    VI_Flood_Alarm := GVL_ALARM.G_Flood_Alarm_Active,
    VI_Security_Alarm := GVL_ALARM.G_Security_Alarm,
    VI_First_Fault_Active := fbSystemHealth.VO_First_Fault_Active,
    VI_First_Fault_Type := fbSystemHealth.VO_First_Fault_Type,
    VI_First_Fault_Source := fbSystemHealth.VO_First_Fault_Source,
    VI_Boiler_Errors := GVL_STATE.G_Boiler_Error,
    VI_Security_Msg := GVL_STATUS.G_Security_Status_Msg,
    VI_Acknowledge_All := GVL_CONFIG.G_HMI_Ack_Alarms OR GVL_COMMAND.G_Reset_Errors,
    VI_Mute_Siren := GVL_CONFIG.G_HMI_Mute_Alarm,
    VIO_Next_Alarm_ID := GVL_ALARM.G_Next_Alarm_ID,
    VO_Global_Critical => GVL_ALARM.G_Global_Critical,
    VO_Global_Warning => GVL_ALARM.G_Global_Warning,
    VO_Siren_Active => GVL_ALARM.G_Global_Siren,
    VO_Active_Count => GVL_ALARM.G_Active_Alarm_Count,
    VO_Unacked_Count => GVL_ALARM.G_Unacked_Alarm_Count,
    VO_Event_Pulse => GVL_STATUS.G_Diagnostics.Alarm_Event_Pulse,
    VO_Event_Code => GVL_STATUS.G_Diagnostics.Alarm_Event_Code,
    VO_Event_Value => GVL_STATUS.G_Diagnostics.Alarm_Event_Value,
    VO_Alarm_List => GVL_ALARM.G_Alarm_List
);

// Command arbitration: OPERATOR > GATEWAY
L_Gateway_Writes_Allowed :=
    NOT GVL_STATUS.G_Diagnostics.Dangerous_Action_Pending_Confirm AND
    NOT GVL_STATUS.G_Diagnostics.Operator_Action_Blocked AND
    NOT GVL_STATUS.G_Diagnostics.User_Access_Denied;

// 13. Интерфейс шлюза (Modbus TCP)
fbGateway(
    VI_System_Time_MS := GVL_STATUS.G_System_Time_MS,
    VI_Local_PLC_Role := SEL(GVL_STATUS.G_Is_Active_PLC, E_PLC_ROLE.ROLE_STANDBY, E_PLC_ROLE.ROLE_ACTIVE),
    VI_Incoming_Command := GVL_GATEWAY.G_Gateway_Command,
    VI_Command_Received := GVL_GATEWAY.G_Gateway_Command_Received,
    VI_FloorHeating_Temps := L_FloorTemps_8,
    VI_Room_Temps := GVL_STATE.G_Room_Temps,
    VI_Zone_Valve_States := L_Zone_Valves_8,
    VI_Manifold_Pressures := GVL_STATE.G_Manifold_Pressures,
    VI_Manifold_Pump_States := GVL_STATE.G_Manifold_Pumps,
    VI_Outdoor_Temp := GVL_STATE.G_Outdoor_Temp,
    VI_Security_Armed := GVL_ALARM.G_Security_Armed,
    VI_Flood_Alarm_Active := GVL_ALARM.G_Flood_Alarm_Active,
    VI_Gas_Alarm_Active := GVL_ALARM.G_Gas_Alarm_Active,
    VI_Fire_Alarm_Active := GVL_ALARM.G_Fire_Alarm_Active,
    VI_Methane_Concentration := GVL_STATE.G_Methane_Sensors[1],
    VI_Lighting_Base_Levels := L_Lighting_32,
    VI_Socket_States := GVL_STATE.G_Socket_States,
    VI_Blinds_Positions := GVL_STATE.G_Blinds_Positions,
    VI_Active_Scenario := GVL_STATUS.G_Current_Scenario,
    VI_Send_2FA_Req := GVL_COMMAND.G_Send_2FA_Req,
    VI_2FA_Code := GVL_COMMAND.G_2FA_Code_Out,
    VI_Allowed_IPs := GVL_CONFIG.G_Allowed_IPs,
    VO_Telegram_Msg => GVL_GATEWAY.G_Gateway_Telegram_Msg,
    VO_Send_Telegram => GVL_GATEWAY.G_Gateway_Send_Telegram,
    VO_HMI_Status_Message => GVL_GATEWAY.G_Gateway_HMI_Status_Message,

    VO_Data_Ready => GVL_GATEWAY.G_Gateway_Data_Ready,
    VO_Modbus_Registers => GVL_GATEWAY.G_Gateway_Modbus_Registers,
    VO_Arm_Req => GVL_COMMAND.G_Arm_Req,
    VO_Disarm_Req => GVL_COMMAND.G_Disarm_Req,
    VO_PIN_Code => GVL_COMMAND.G_PIN_Code,
    VO_RFID_Tag => GVL_COMMAND.G_RFID_Tag,
    VO_2FA_Code_In => GVL_COMMAND.G_2FA_Code_In,
    VO_Lighting_Override => GVL_COMMAND.G_Lighting_Override,
    VO_Blinds_Override => GVL_COMMAND.G_Blinds_Override,
    VO_Socket_Override => GVL_COMMAND.G_Socket_Override,
    VO_Reset_Errors_Req => GVL_COMMAND.G_Reset_Errors
);

IF L_Gateway_Writes_Allowed AND
   fbGateway.VO_Set_Scenario_Req AND
   ((GVL_STATE.G_System_Mode = E_System_Operating_Mode.MODE_NORMAL) OR
    (GVL_STATE.G_System_Mode = E_System_Operating_Mode.MODE_DEGRADED)) THEN
    GVL_COMMAND.G_Scenario_Request := fbGateway.VO_Target_Scenario;
END_IF;

IF L_Gateway_Writes_Allowed AND
   fbGateway.VO_Set_Temp_Req AND
   (GVL_STATE.G_System_Mode = E_System_Operating_Mode.MODE_NORMAL) THEN
    GVL_CONFIG.G_HMI_FloorHeating_Configs[fbGateway.VO_Target_Zone].design_temp := fbGateway.VO_Target_Temp;
END_IF;

IF L_Gateway_Writes_Allowed AND
   fbGateway.VO_Set_Vent_Req AND
   (GVL_STATE.G_System_Mode = E_System_Operating_Mode.MODE_NORMAL) THEN
    GVL_CONFIG.G_HMI_Vent_Global_Config.default_supply_speed := fbGateway.VO_Target_Vent_Speed;
END_IF;

IF L_Gateway_Writes_Allowed AND
   fbGateway.VO_Set_Config_Req AND
   (GVL_STATE.G_System_Mode = E_System_Operating_Mode.MODE_NORMAL) THEN
    GVL_CONFIG.G_HMI_Apply_Settings := TRUE;
END_IF;

IF L_Gateway_Writes_Allowed AND
   fbGateway.VO_Sync_Time_Req AND
   (GVL_STATE.G_System_Mode = E_System_Operating_Mode.MODE_NORMAL) THEN
    GVL_STATUS.G_Time_Of_Day_MS := fbGateway.VO_New_Time_MS;
END_IF;

// ================= COMMAND GATE (FINAL) =================
IF GVL_STATE.G_System_Mode = E_System_Operating_Mode.MODE_SAFE_STOP THEN

    // Блокируем ВСЕ опасные команды после Gateway
    GVL_COMMAND.G_Scenario_Request := 0;

    FOR L_i := 1 TO 32 DO
        GVL_COMMAND.G_Lighting_Override[L_i] := BYTE#0;
        GVL_COMMAND.G_Blinds_Override[L_i] := BYTE#0;
        GVL_COMMAND.G_Socket_Override[L_i] := FALSE;
    END_FOR;

    // НЕ блокируем:
    // G_Reset_Errors
    // acknowledge / безопасность

END_IF;
// =======================================================

// 14. Менеджер NVRAM
IF NOT L_Config_Loaded THEN
    L_NVRAM_Cmd := 2; // READ
    L_NVRAM_Offset := 0;
    L_Config_Loaded := TRUE;
ELSIF GVL_CONFIG.G_HMI_Apply_Settings THEN
    L_NVRAM_Cmd := 1; // WRITE
    L_NVRAM_Offset := 0;
    GVL_CONFIG.G_HMI_Apply_Settings := FALSE;
ELSE
    L_NVRAM_Cmd := 0;
END_IF;

// fbNVRAMManager(
//     VI_Command := L_NVRAM_Cmd,
//     VI_Offset := L_NVRAM_Offset,
// // //     VI_System_Time_MS := GVL_STATUS.G_System_Time_MS,
//     VI_Operator_ID := 'SYSTEM',
//     VI_IsActivePLC := GVL_STATUS.G_Is_Active_PLC,
//     VI_TwoPersonConfirmation := FALSE,
//     VO_Done => L_NVRAM_Done,
//     VO_Error => L_NVRAM_Err,
//     VO_ErrorID => L_NVRAM_ErrID
// );

// 15. Черный ящик
L_BB_Record.Timestamp := GVL_STATUS.G_System_Time_MS;
L_BB_Record.PLC_Active_ID := GVL_STATUS.G_PLC_ID;
L_BB_Record.Gas_Methane_LEL := GVL_STATE.G_Methane_Sensors[1];
L_BB_Record.Gas_CO_PPM := GVL_STATE.G_CO_Sensors[1];
L_BB_Record.Flood_Active := GVL_ALARM.G_Flood_Alarm_Active;
L_BB_Record.Fire_Active := GVL_ALARM.G_Fire_Alarm_Active;
L_BB_Record.Valve_Gas_Status := SEL(GVL_COMMAND.G_Gas_Valve_Close, BYTE#0, BYTE#1);
L_BB_Record.Valve_Water_Status := SEL((GVL_COMMAND.G_Close_Valve_35 OR GVL_COMMAND.G_Close_Valve_36), BYTE#0, BYTE#1);

L_BB_Record.System_Mode := TO_BYTE(TO_INT(GVL_STATE.G_System_Mode));
L_BB_Record.First_Fault_Type := TO_BYTE(TO_INT(fbSystemHealth.VO_First_Fault_Type));
L_BB_Record.First_Fault_Source := TO_BYTE(TO_INT(fbSystemHealth.VO_First_Fault_Source));
L_BB_Record.First_Fault_Active := fbSystemHealth.VO_First_Fault_Active;
L_BB_Record.System_Severity := TO_BYTE(TO_INT(fbSystemHealth.VO_System_Severity));
L_BB_Record.Root_Cause := TO_BYTE(TO_INT(fbSystemHealth.VO_Root_Cause));
L_BB_Record.Watchdog_Fault := fbWatchdog.VO_Watchdog_Fault;

L_BB_Freeze := GVL_ALARM.G_Gas_Alarm_Active OR GVL_ALARM.G_Fire_Alarm_Active OR GVL_ALARM.G_Flood_Alarm_Active OR fbSystemHealth.VO_First_Fault_Active;

fbBlackBox(
    VI_Current_Data := L_BB_Record,
    VI_Freeze := L_BB_Freeze
);

// 15.1. Менеджер истории / diagnostics bridge
L_History_Write_Event := FALSE;
L_History_Event.timestamp_ms := GVL_STATUS.G_System_Time_MS;
L_History_Event.event_code := 0;
L_History_Event.event_value := 0.0;
L_History_Event.unit := 0;
L_History_Event.zone_id := 0;
L_History_Event.operator_id := 'SYSTEM';
L_History_Event.priority := E_ALERT_PRIORITY.ALERT_PRIORITY_HIGH;

IF GVL_STATE.G_System_Mode <> L_Last_System_Mode THEN
    L_History_Write_Event := TRUE;
    L_History_Event.event_code := 1101; // System mode transition
    L_History_Event.event_value := TO_REAL(TO_INT(GVL_STATE.G_System_Mode));
    L_History_Event.unit := 1; // system mode domain
    L_History_Event.zone_id := 0;
    IF GVL_STATE.G_System_Mode = E_System_Operating_Mode.MODE_NORMAL THEN
        L_History_Event.priority := E_ALERT_PRIORITY.ALERT_PRIORITY_HIGH;
    ELSE
        L_History_Event.priority := E_ALERT_PRIORITY.ALERT_PRIORITY_HIGH;
    END_IF;
    L_Last_System_Mode := GVL_STATE.G_System_Mode;

ELSIF fbSystemHealth.VO_Root_Cause <> L_Last_Root_Cause THEN
    L_History_Write_Event := TRUE;
    L_History_Event.event_code := 1102; // Root cause changed
    L_History_Event.event_value := TO_REAL(TO_INT(fbSystemHealth.VO_Root_Cause));
    L_History_Event.unit := 2; // root cause enum domain
    L_History_Event.zone_id := TO_BYTE(fbSystemHealth.VO_First_Fault_Source);
    L_History_Event.priority := E_ALERT_PRIORITY.ALERT_PRIORITY_HIGH;
    L_Last_Root_Cause := fbSystemHealth.VO_Root_Cause;

ELSIF fbSystemHealth.VO_First_Fault_Source <> L_Last_First_Fault_Source THEN
    L_History_Write_Event := TRUE;
    L_History_Event.event_code := 1103; // First fault source changed
    L_History_Event.event_value := TO_REAL(fbSystemHealth.VO_First_Fault_Source);
    L_History_Event.unit := 3; // root cause source domain
    L_History_Event.zone_id := TO_BYTE(fbSystemHealth.VO_First_Fault_Source);
    L_History_Event.priority := E_ALERT_PRIORITY.ALERT_PRIORITY_HIGH;
    L_Last_First_Fault_Source := fbSystemHealth.VO_First_Fault_Source;

ELSIF GVL_STATUS.G_Current_Scenario <> GVL_STATUS.G_Previous_Scenario THEN
    L_History_Write_Event := TRUE;
    L_History_Event.event_code := 1001; // Scenario transition
    L_History_Event.event_value := TO_REAL(GVL_STATUS.G_Current_Scenario);
    L_History_Event.unit := 4; // scenario domain
    L_History_Event.zone_id := 0;
    L_History_Event.priority := E_ALERT_PRIORITY.ALERT_PRIORITY_HIGH;
    GVL_STATUS.G_Previous_Scenario := GVL_STATUS.G_Current_Scenario;

ELSIF GVL_STATUS.G_Diagnostics.Alarm_Event_Pulse THEN
    L_History_Write_Event := TRUE;
    L_History_Event.event_code := TO_WORD(GVL_STATUS.G_Diagnostics.Alarm_Event_Code);
    L_History_Event.event_value := GVL_STATUS.G_Diagnostics.Alarm_Event_Value;
    L_History_Event.unit := 10; // alarm lifecycle domain
    L_History_Event.zone_id := 0;
    L_History_Event.priority := E_ALERT_PRIORITY.ALERT_PRIORITY_HIGH;

ELSIF GVL_STATUS.G_Diagnostics.Operator_Journal_Event_Seq <> L_Last_Operator_Journal_Seq THEN
    L_History_Write_Event := TRUE;
    L_History_Event.event_code := 1301; // Operator journal event
    L_History_Event.event_value := TO_REAL(GVL_STATUS.G_Diagnostics.Operator_Journal_Event_Seq);
    L_History_Event.unit := 20; // operator journal domain
    L_History_Event.zone_id := 0;
    L_History_Event.priority := E_ALERT_PRIORITY.ALERT_PRIORITY_HIGH;
    L_Last_Operator_Journal_Seq := GVL_STATUS.G_Diagnostics.Operator_Journal_Event_Seq;
END_IF;

// --- History anti-flood / dedup ---
IF L_History_Write_Event THEN
    IF (L_History_Event.event_code = L_Last_Event_Code)
       AND (ABS(L_History_Event.event_value - L_Last_Event_Value) < 0.001)
       AND (GVL_STATUS.G_System_Time_MS - L_Last_Event_Time_MS < 5000) THEN
        L_History_Write_Event := FALSE;
    ELSE
        L_Last_Event_Code := L_History_Event.event_code;
        L_Last_Event_Value := L_History_Event.event_value;
        L_Last_Event_Time_MS := GVL_STATUS.G_System_Time_MS;
    END_IF;
END_IF;

fbHistoryManager(
    VI_System_Time_MS := GVL_STATUS.G_System_Time_MS,
    VI_Write_Event := L_History_Write_Event,
    VI_Event := L_History_Event
);

// HMI maintenance mode control (confirmation-aware)
IF GVL_COMMAND.CMD_Dangerous_Action_Confirm THEN
    FOR L_i := 1 TO GVL_CONSTANTS.C_MAX_MANIFOLDS DO
        GVL_CONFIG.G_Manifold_Pump_In_Service[L_i] := GVL_COMMAND.CMD_Set_Manifold_Pump_In_Service[L_i];
    END_FOR;
    GVL_CONFIG.G_DHW_Heating_Pump_In_Service := GVL_COMMAND.CMD_Set_DHW_Heating_Pump_In_Service;
    GVL_CONFIG.G_DHW_Circ_Pump_In_Service := GVL_COMMAND.CMD_Set_DHW_Circ_Pump_In_Service;
END_IF;

// Dangerous action confirmation flow
IF GVL_COMMAND.CMD_Dangerous_Action_Request THEN
    L_Dangerous_Action_Armed := TRUE;
    L_Dangerous_Action_Deadline_MS := GVL_STATUS.G_System_Time_MS + 15000;
    GVL_STATUS.G_Diagnostics.Dangerous_Action_Pending_Confirm := TRUE;
    GVL_STATUS.G_Diagnostics.Dangerous_Action_Confirm_Deadline_MS := L_Dangerous_Action_Deadline_MS;
    GVL_STATUS.G_Diagnostics.Dangerous_Action_Confirm_Text := 'Подтвердите опасное действие в течение 15 секунд';
END_IF;
IF L_Dangerous_Action_Armed AND (GVL_STATUS.G_System_Time_MS > L_Dangerous_Action_Deadline_MS) THEN
    L_Dangerous_Action_Armed := FALSE;
    GVL_STATUS.G_Diagnostics.Dangerous_Action_Pending_Confirm := FALSE;
    GVL_STATUS.G_Diagnostics.Dangerous_Action_Confirm_Text := 'Окно подтверждения истекло';
END_IF;
IF GVL_COMMAND.CMD_Dangerous_Action_Confirm AND L_Dangerous_Action_Armed THEN
    L_Dangerous_Action_Armed := FALSE;
    GVL_STATUS.G_Diagnostics.Dangerous_Action_Pending_Confirm := FALSE;
    GVL_STATUS.G_Diagnostics.Dangerous_Action_Confirm_Text := 'Опасное действие подтверждено оператором';
END_IF;

// Access level enforcement for dangerous actions
GVL_STATUS.G_Diagnostics.User_Access_Level_Active := GVL_COMMAND.CMD_User_Access_Level;
GVL_STATUS.G_Diagnostics.User_Access_Denied := FALSE;
GVL_STATUS.G_Diagnostics.User_Access_Deny_Reason := '';
IF GVL_COMMAND.CMD_Dangerous_Action_Request OR GVL_COMMAND.CMD_Dangerous_Action_Confirm THEN
    IF GVL_COMMAND.CMD_User_Access_Level < 2 THEN
        GVL_STATUS.G_Diagnostics.User_Access_Denied := TRUE;
        GVL_STATUS.G_Diagnostics.User_Access_Deny_Reason := 'Недостаточный уровень доступа для опасного действия';
        GVL_STATUS.G_Diagnostics.Operator_Action_Blocked := TRUE;
        GVL_STATUS.G_Diagnostics.Operator_Block_Reason := 'Требуется уровень ENGINEER для опасного действия';
        GVL_STATUS.G_Diagnostics.Dangerous_Action_Pending_Confirm := FALSE;
        GVL_STATUS.G_Diagnostics.Dangerous_Action_Confirm_Text := 'Доступ запрещён: требуется уровень ENGINEER';
    END_IF;
END_IF;

// Hard revert for forbidden operator actions
IF GVL_STATUS.G_Diagnostics.Operator_Action_Blocked THEN
    FOR L_i := 1 TO GVL_CONSTANTS.C_MAX_MANIFOLDS DO
        IF NOT GVL_CONFIG.G_Manifold_Pump_In_Service[L_i] THEN
            GVL_CONFIG.G_Manifold_Pump_In_Service[L_i] := TRUE;
        END_IF;
    END_FOR;
    IF NOT GVL_CONFIG.G_DHW_Heating_Pump_In_Service THEN
        GVL_CONFIG.G_DHW_Heating_Pump_In_Service := TRUE;
    END_IF;
    IF NOT GVL_CONFIG.G_DHW_Circ_Pump_In_Service THEN
        GVL_CONFIG.G_DHW_Circ_Pump_In_Service := TRUE;
    END_IF;
    GVL_STATUS.G_Diagnostics.Operator_Last_Forbidden_Action := GVL_STATUS.G_Diagnostics.Operator_Block_Reason;
END_IF;

// Operator action journal
IF GVL_STATUS.G_Diagnostics.Operator_Action_Blocked AND NOT L_Last_Operator_Blocked THEN
    GVL_STATUS.G_Diagnostics.Operator_Journal_Event_Seq := GVL_STATUS.G_Diagnostics.Operator_Journal_Event_Seq + 1;
END_IF;
L_Last_Operator_Blocked := GVL_STATUS.G_Diagnostics.Operator_Action_Blocked;
IF GVL_CONFIG.G_DHW_Heating_Pump_In_Service <> L_Last_DHW_Heating_In_Service THEN
    GVL_STATUS.G_Diagnostics.Operator_Journal_Event_Seq := GVL_STATUS.G_Diagnostics.Operator_Journal_Event_Seq + 1;
    IF GVL_CONFIG.G_DHW_Heating_Pump_In_Service THEN
        GVL_STATUS.G_Diagnostics.Maintenance_Last_Action := 'Насос загрузки ГВС возвращён из ТО';
    ELSE
        GVL_STATUS.G_Diagnostics.Maintenance_Last_Action := 'Насос загрузки ГВС выведен в ТО';
    END_IF;
END_IF;
L_Last_DHW_Heating_In_Service := GVL_CONFIG.G_DHW_Heating_Pump_In_Service;
IF GVL_CONFIG.G_DHW_Circ_Pump_In_Service <> L_Last_DHW_Circ_In_Service THEN
    GVL_STATUS.G_Diagnostics.Operator_Journal_Event_Seq := GVL_STATUS.G_Diagnostics.Operator_Journal_Event_Seq + 1;
    IF GVL_CONFIG.G_DHW_Circ_Pump_In_Service THEN
        GVL_STATUS.G_Diagnostics.Maintenance_Last_Action := 'Насос рециркуляции ГВС возвращён из ТО';
    ELSE
        GVL_STATUS.G_Diagnostics.Maintenance_Last_Action := 'Насос рециркуляции ГВС выведен в ТО';
    END_IF;
END_IF;
L_Last_DHW_Circ_In_Service := GVL_CONFIG.G_DHW_Circ_Pump_In_Service;
IF GVL_STATUS.G_Diagnostics.Operator_Journal_Event_Seq <> GVL_STATUS.G_Diagnostics.Operator_Journal_Last_Seq THEN
    GVL_STATUS.G_Diagnostics.Operator_Journal_3 := GVL_STATUS.G_Diagnostics.Operator_Journal_2;
    GVL_STATUS.G_Diagnostics.Operator_Journal_2 := GVL_STATUS.G_Diagnostics.Operator_Journal_1;
    IF GVL_STATUS.G_Diagnostics.Operator_Last_Forbidden_Action <> '' THEN
        GVL_STATUS.G_Diagnostics.Operator_Journal_1 := GVL_STATUS.G_Diagnostics.Operator_Last_Forbidden_Action;
    ELSE
        GVL_STATUS.G_Diagnostics.Operator_Journal_1 := GVL_STATUS.G_Diagnostics.Maintenance_Last_Action;
    END_IF;
    GVL_STATUS.G_Diagnostics.Operator_Journal_Last_Seq := GVL_STATUS.G_Diagnostics.Operator_Journal_Event_Seq;
END_IF;

// ========================================
// CoreKernel live observer (diagnostic only)
// ========================================
// fbCoreKernelObserver disabled temporarily

// >>> BULK_SYNC_ANCHOR: PRG_System <<<
